LIN {X 0,Y 328.943,Z 502.897,A -85,B 0,C 180,E1 -15636.784,E2 -15636.784} C_VEL
LIN {X 0,Y 327.301,Z 513.257,A -85,B 0,C 180,E1 -15637.783,E2 -15637.783} C_VEL
LIN {X 0,Y 325.235,Z 524.397,A -85,B 0,C 180,E1 -15639.111,E2 -15639.111} C_VEL
LIN {X 0,Y 323.008,Z 534.604,A -85,B 0,C 180,E1 -15640.621,E2 -15640.621} C_VEL
LIN {X 0,Y 320.683,Z 544.507,A -85,B 0,C 180,E1 -15642.462,E2 -15642.462} C_VEL
LIN {X 0,Y 318.696,Z 552.395,A -85,B 0,C 180,E1 -15644.327,E2 -15644.327} C_VEL
LIN {X 0,Y 317.23,Z 557.815,A -85,B 0,C 180,E1 -15645.895,E2 -15645.895} C_VEL
LIN {X 0,Y 315.687,Z 563.068,A -85,B 0,C 180,E1 -15647.79,E2 -15647.79} C_VEL
LIN {X 0,Y 314.434,Z 567.146,A -85,B 0,C 180,E1 -15649.699,E2 -15649.699} C_VEL
LIN {X 0,Y 313.55,Z 569.293,A -85,B 0,C 180,E1 -15650.973,E2 -15650.973} C_VEL
LIN {X 0,Y 313.019,Z 570.939,A -85,B 0,C 180,E1 -15652.258,E2 -15652.258} C_VEL
LIN {X 0,Y 312.547,Z 572.122,A -85,B 0,C 180,E1 -15653.544,E2 -15653.544} C_VEL
LIN {X 0,Y 312.335,Z 572.873,A -85,B 0,C 180,E1 -15654.836,E2 -15654.836} C_VEL
LIN {X 0,Y 312.032,Z 573.237,A -85,B 0,C 180,E1 -15656.125,E2 -15656.125} C_VEL
LIN {X 0,Y 311.617,Z 573.155,A -85,B 0,C 180,E1 -15657.415,E2 -15657.415} C_VEL
LIN {X 0,Y 311.355,Z 572.635,A -85,B 0,C 180,E1 -15658.706,E2 -15658.706} C_VEL
LIN {X 0,Y 311.243,Z 571.699,A -85,B 0,C 180,E1 -15660,E2 -15660} C_VEL
LIN {X 0,Y 311.196,Z 570.316,A -85,B 0,C 180,E1 -15661.294,E2 -15661.294} C_VEL
LIN {X 0,Y 311.223,Z 567.384,A -85,B 0,C 180,E1 -15663.236,E2 -15663.236} C_VEL
LIN {X 0,Y 311.418,Z 563.364,A -85,B 0,C 180,E1 -15665.179,E2 -15665.179} C_VEL
LIN {X 0,Y 311.687,Z 557.186,A -85,B 0,C 180,E1 -15667.436,E2 -15667.436} C_VEL
LIN {X 0,Y 312.083,Z 550.339,A -85,B 0,C 180,E1 -15669.396,E2 -15669.396} C_VEL
LIN {X 0,Y 312.706,Z 541.811,A -85,B 0,C 180,E1 -15671.341,E2 -15671.341} C_VEL
LIN {X 0,Y 313.329,Z 533.139,A -85,B 0,C 180,E1 -15672.962,E2 -15672.962} C_VEL
LIN {X 0,Y 314.181,Z 522.592,A -85,B 0,C 180,E1 -15674.575,E2 -15674.575} C_VEL
LIN {X 0,Y 315.066,Z 510.768,A -85,B 0,C 180,E1 -15676.027,E2 -15676.027} C_VEL
LIN {X 0,Y 315.637,Z 499.309,A -85,B 0,C 180,E1 -15677.159,E2 -15677.159} C_VEL
LIN {X 0,Y 316.398,Z 485.475,A -85,B 0,C 180,E1 -15678.202,E2 -15678.202} C_VEL
LIN {X 0,Y 317.017,Z 472.382,A -85,B 0,C 180,E1 -15678.918,E2 -15678.918} C_VEL
LIN {X 0,Y 317.51,Z 455.689,A -85,B 0,C 180,E1 -15679.517,E2 -15679.517} C_VEL
LIN {X 0,Y 319.541,Z 389.489,A -85,B 0,C 180,E1 -15681.639,E2 -15681.639} C_VEL
LIN {X 0,Y 312.571,Z 367.548,A -85,B 0,C 180,E1 -15682.686,E2 -15682.686} C_VEL
LIN {X 0,Y 312.608,Z 367.544,A -85,B 0,C 180,E1 -15685.935,E2 -15685.935} C_VEL
LIN {X 0,Y 312.55,Z 367.55,A -85,B 0,C 180,E1 -15689.649,E2 -15689.649} C_VEL
LIN {X 0,Y 312.524,Z 367.553,A -85,B 0,C 180,E1 -15693.688,E2 -15693.688} C_VEL
LIN {X 0,Y 312.53,Z 367.552,A -85,B 0,C 180,E1 -15697.384,E2 -15697.384} C_VEL
LIN {X 0,Y 312.494,Z 367.558,A -85,B 0,C 180,E1 -15700.708,E2 -15700.708} C_VEL
LIN {X 0,Y 312.456,Z 367.566,A -85,B 0,C 180,E1 -15704.209,E2 -15704.209} C_VEL
LIN {X 0,Y 312.488,Z 367.56,A -85,B 0,C 180,E1 -15707.918,E2 -15707.918} C_VEL
LIN {X 0,Y 312.539,Z 367.553,A -85,B 0,C 180,E1 -15711.91,E2 -15711.91} C_VEL
LIN {X 0,Y 312.51,Z 367.556,A -85,B 0,C 180,E1 -15715.789,E2 -15715.789} C_VEL
LIN {X 0,Y 312.524,Z 367.553,A -85,B 0,C 180,E1 -15718.853,E2 -15718.853} C_VEL
LIN {X 0,Y 312.574,Z 367.549,A -85,B 0,C 180,E1 -15721.823,E2 -15721.823} C_VEL
LIN {X 0,Y 312.589,Z 367.545,A -85,B 0,C 180,E1 -15724.71,E2 -15724.71} C_VEL
LIN {X 0,Y 312.591,Z 367.545,A -85,B 0,C 180,E1 -15727.528,E2 -15727.528} C_VEL
LIN {X 0,Y 312.642,Z 367.54,A -85,B 0,C 180,E1 -15731.655,E2 -15731.655} C_VEL
LIN {X 0,Y 312.697,Z 367.533,A -85,B 0,C 180,E1 -15735.685,E2 -15735.685} C_VEL
LIN {X 0,Y 312.701,Z 367.532,A -85,B 0,C 180,E1 -15739.64,E2 -15739.64} C_VEL
LIN {X 0,Y 312.855,Z 367.515,A -85,B 0,C 180,E1 -15742.252,E2 -15742.252} C_VEL
LIN {X 0,Y 312.718,Z 367.528,A -85,B 0,C 180,E1 -15744.841,E2 -15744.841} C_VEL
LIN {X 0,Y 312.993,Z 367.495,A -85,B 0,C 180,E1 -15748.712,E2 -15748.712} C_VEL
LIN {X 0,Y 313.122,Z 367.484,A -85,B 0,C 180,E1 -15749.999,E2 -15749.999} C_VEL
LIN {X 0,Y 312.94,Z 367.502,A -85,B 0,C 180,E1 -15752.573,E2 -15752.573} C_VEL
LIN {X 0,Y 312.911,Z 367.506,A -85,B 0,C 180,E1 -15756.446,E2 -15756.446} C_VEL
LIN {X 0,Y 312.787,Z 367.52,A -85,B 0,C 180,E1 -15759.048,E2 -15759.048} C_VEL
LIN {X 0,Y 312.633,Z 367.539,A -85,B 0,C 180,E1 -15762.989,E2 -15762.989} C_VEL
LIN {X 0,Y 312.637,Z 367.541,A -85,B 0,C 180,E1 -15765.648,E2 -15765.648} C_VEL
LIN {X 0,Y 312.629,Z 367.54,A -85,B 0,C 180,E1 -15769.235,E2 -15769.235} C_VEL
LIN {X 0,Y 312.543,Z 367.55,A -85,B 0,C 180,E1 -15772.788,E2 -15772.788} C_VEL
LIN {X 0,Y 312.6,Z 367.548,A -85,B 0,C 180,E1 -15775.934,E2 -15775.934} C_VEL
LIN {X 0,Y 312.542,Z 367.554,A -85,B 0,C 180,E1 -15779.648,E2 -15779.648} C_VEL
LIN {X 0,Y 312.515,Z 367.558,A -85,B 0,C 180,E1 -15783.688,E2 -15783.688} C_VEL
LIN {X 0,Y 312.548,Z 367.551,A -85,B 0,C 180,E1 -15787.38,E2 -15787.38} C_VEL
LIN {X 0,Y 312.529,Z 367.552,A -85,B 0,C 180,E1 -15790.701,E2 -15790.701} C_VEL
LIN {X 0,Y 312.589,Z 367.546,A -85,B 0,C 180,E1 -15794.183,E2 -15794.183} C_VEL
LIN {X 0,Y 312.55,Z 367.553,A -85,B 0,C 180,E1 -15797.903,E2 -15797.903} C_VEL
LIN {X 0,Y 312.55,Z 367.553,A -85,B 0,C 180,E1 -15801.904,E2 -15801.904} C_VEL
LIN {X 0,Y 312.498,Z 367.56,A -85,B 0,C 180,E1 -15805.789,E2 -15805.789} C_VEL
LIN {X 0,Y 312.515,Z 367.554,A -85,B 0,C 180,E1 -15808.853,E2 -15808.853} C_VEL
LIN {X 0,Y 312.576,Z 367.55,A -85,B 0,C 180,E1 -15811.825,E2 -15811.825} C_VEL
LIN {X 0,Y 312.577,Z 367.546,A -85,B 0,C 180,E1 -15814.71,E2 -15814.71} C_VEL
LIN {X 0,Y 312.578,Z 367.55,A -85,B 0,C 180,E1 -15817.528,E2 -15817.528} C_VEL
LIN {X 0,Y 312.616,Z 367.542,A -85,B 0,C 180,E1 -15821.173,E2 -15821.173} C_VEL
LIN {X 0,Y 311.964,Z 367.628,A -85,B 0,C 180,E1 -15822.249,E2 -15822.249} C_VEL
LIN {X 0,Y 309.133,Z 367.983,A -85,B 0,C 180,E1 -15824.002,E2 -15824.002} C_VEL
LIN {X 0,Y 306.716,Z 368.281,A -85,B 0,C 180,E1 -15825.423,E2 -15825.423} C_VEL
LIN {X 0,Y 305.666,Z 368.407,A -85,B 0,C 180,E1 -15826.523,E2 -15826.523} C_VEL
LIN {X 0,Y 305.573,Z 368.417,A -85,B 0,C 180,E1 -15826.895,E2 -15826.895} C_VEL
LIN {X 0,Y 305.787,Z 368.394,A -85,B 0,C 180,E1 -15831.208,E2 -15831.208} C_VEL
LIN {X 0,Y 305.843,Z 368.389,A -85,B 0,C 180,E1 -15833.403,E2 -15833.403} C_VEL
LIN {X 0,Y 305.89,Z 368.383,A -85,B 0,C 180,E1 -15837.366,E2 -15837.366} C_VEL
LIN {X 0,Y 306.064,Z 368.358,A -85,B 0,C 180,E1 -15840,E2 -15840} C_VEL
LIN {X 0,Y 305.879,Z 368.38,A -85,B 0,C 180,E1 -15842.634,E2 -15842.634} C_VEL
LIN {X 0,Y 305.846,Z 368.385,A -85,B 0,C 180,E1 -15846.598,E2 -15846.598} C_VEL
LIN {X 0,Y 305.727,Z 368.403,A -85,B 0,C 180,E1 -15849.26,E2 -15849.26} C_VEL
LIN {X 0,Y 305.582,Z 368.421,A -85,B 0,C 180,E1 -15853.296,E2 -15853.296} C_VEL
LIN {X 0,Y 305.585,Z 368.418,A -85,B 0,C 180,E1 -15856.021,E2 -15856.021} C_VEL
LIN {X 0,Y 305.568,Z 368.424,A -85,B 0,C 180,E1 -15859.446,E2 -15859.446} C_VEL
LIN {X 0,Y 305.482,Z 368.432,A -85,B 0,C 180,E1 -15863.042,E2 -15863.042} C_VEL
LIN {X 0,Y 305.517,Z 368.425,A -85,B 0,C 180,E1 -15866.22,E2 -15866.22} C_VEL
LIN {X 0,Y 305.48,Z 368.432,A -85,B 0,C 180,E1 -15869.048,E2 -15869.048} C_VEL
LIN {X 0,Y 305.434,Z 368.437,A -85,B 0,C 180,E1 -15871.954,E2 -15871.954} C_VEL
LIN {X 0,Y 305.456,Z 368.437,A -85,B 0,C 180,E1 -15875.114,E2 -15875.114} C_VEL
LIN {X 0,Y 305.489,Z 368.429,A -85,B 0,C 180,E1 -15878.541,E2 -15878.541} C_VEL
LIN {X 0,Y 305.516,Z 368.426,A -85,B 0,C 180,E1 -15882.601,E2 -15882.601} C_VEL
LIN {X 0,Y 305.529,Z 368.423,A -85,B 0,C 180,E1 -15886.366,E2 -15886.366} C_VEL
LIN {X 0,Y 305.495,Z 368.429,A -85,B 0,C 180,E1 -15889.901,E2 -15889.901} C_VEL
LIN {X 0,Y 305.498,Z 368.429,A -85,B 0,C 180,E1 -15893.628,E2 -15893.628} C_VEL
LIN {X 0,Y 305.54,Z 368.505,A -85,B 0,C 180,E1 -15896.939,E2 -15896.939} C_VEL
LIN {X 0,Y 308.728,Z 384.104,A -85,B 0,C 180,E1 -15901.072,E2 -15901.072} C_VEL
LIN {X 0,Y 309.707,Z 390.276,A -85,B 0,C 180,E1 -15902.649,E2 -15902.649} C_VEL
LIN {X 0,Y 308.052,Z 404.751,A -85,B 0,C 180,E1 -15906.14,E2 -15906.14} C_VEL
LIN {X 0,Y 307.818,Z 407.252,A -85,B 0,C 180,E1 -15906.719,E2 -15906.719} C_VEL
LIN {X 0,Y 309.835,Z 432.681,A -85,B 0,C 180,E1 -15907.693,E2 -15907.693} C_VEL
LIN {X 0,Y 311.778,Z 451.87,A -85,B 0,C 180,E1 -15908.433,E2 -15908.433} C_VEL
LIN {X 0,Y 309.786,Z 517.337,A -85,B 0,C 180,E1 -15910.667,E2 -15910.667} C_VEL
LIN {X 0,Y 309.008,Z 530.335,A -85,B 0,C 180,E1 -15911.349,E2 -15911.349} C_VEL
LIN {X 0,Y 308.149,Z 542.629,A -85,B 0,C 180,E1 -15912.241,E2 -15912.241} C_VEL
LIN {X 0,Y 307.335,Z 554.72,A -85,B 0,C 180,E1 -15913.392,E2 -15913.392} C_VEL
LIN {X 0,Y 306.479,Z 565.586,A -85,B 0,C 180,E1 -15914.687,E2 -15914.687} C_VEL
LIN {X 0,Y 305.7,Z 575.858,A -85,B 0,C 180,E1 -15916.202,E2 -15916.202} C_VEL
LIN {X 0,Y 304.994,Z 585.89,A -85,B 0,C 180,E1 -15918.032,E2 -15918.032} C_VEL
LIN {X 0,Y 304.522,Z 593.338,A -85,B 0,C 180,E1 -15919.698,E2 -15919.698} C_VEL
LIN {X 0,Y 304.314,Z 600.602,A -85,B 0,C 180,E1 -15921.702,E2 -15921.702} C_VEL
LIN {X 0,Y 304.237,Z 606.711,A -85,B 0,C 180,E1 -15923.857,E2 -15923.857} C_VEL
LIN {X 0,Y 304.227,Z 611.32,A -85,B 0,C 180,E1 -15926.028,E2 -15926.028} C_VEL
LIN {X 0,Y 304.239,Z 613.406,A -85,B 0,C 180,E1 -15927.354,E2 -15927.354} C_VEL
LIN {X 0,Y 304.424,Z 615.02,A -85,B 0,C 180,E1 -15928.679,E2 -15928.679} C_VEL
LIN {X 0,Y 304.4,Z 616.15,A -85,B 0,C 180,E1 -15930.002,E2 -15930.002} C_VEL
LIN {X 0,Y 304.147,Z 616.77,A -85,B 0,C 180,E1 -15931.326,E2 -15931.326} C_VEL
LIN {X 0,Y 304.008,Z 616.934,A -85,B 0,C 180,E1 -15932.652,E2 -15932.652} C_VEL
LIN {X 0,Y 303.856,Z 616.667,A -85,B 0,C 180,E1 -15933.98,E2 -15933.98} C_VEL
LIN {X 0,Y 303.815,Z 615.504,A -85,B 0,C 180,E1 -15935.901,E2 -15935.901} C_VEL
LIN {X 0,Y 304.016,Z 612.303,A -85,B 0,C 180,E1 -15938.644,E2 -15938.644} C_VEL
LIN {X 0,Y 304.52,Z 608.766,A -85,B 0,C 180,E1 -15940.641,E2 -15940.641} C_VEL
LIN {X 0,Y 305.392,Z 604.144,A -85,B 0,C 180,E1 -15942.63,E2 -15942.63} C_VEL
LIN {X 0,Y 306.856,Z 597.249,A -85,B 0,C 180,E1 -15944.933,E2 -15944.933} C_VEL
LIN {X 0,Y 308.362,Z 590.584,A -85,B 0,C 180,E1 -15946.723,E2 -15946.723} C_VEL
LIN {X 0,Y 310.363,Z 582.557,A -85,B 0,C 180,E1 -15948.484,E2 -15948.484} C_VEL
LIN {X 0,Y 312.535,Z 573.888,A -85,B 0,C 180,E1 -15950.057,E2 -15950.057} C_VEL
LIN {X 0,Y 314.949,Z 563.526,A -85,B 0,C 180,E1 -15951.606,E2 -15951.606} C_VEL
LIN {X 0,Y 317.789,Z 550.815,A -85,B 0,C 180,E1 -15953.114,E2 -15953.114} C_VEL
LIN {X 0,Y 320.028,Z 539.948,A -85,B 0,C 180,E1 -15954.144,E2 -15954.144} C_VEL
LIN {X 0,Y 322.595,Z 526.17,A -85,B 0,C 180,E1 -15955.141,E2 -15955.141} C_VEL
LIN {X 0,Y 324.642,Z 512.058,A -85,B 0,C 180,E1 -15955.916,E2 -15955.916} C_VEL
LIN {X 0,Y 328.062,Z 476.175,A -85,B 0,C 180,E1 -15957.317,E2 -15957.317} C_VEL
LIN {X 0,Y 329.941,Z 456.205,A -85,B 0,C 180,E1 -15958.101,E2 -15958.101} C_VEL
LIN {X 0,Y 329.581,Z 444.672,A -85,B 0,C 180,E1 -15958.851,E2 -15958.851} C_VEL
LIN {X 0,Y 328.161,Z 430.684,A -85,B 0,C 180,E1 -15960.026,E2 -15960.026} C_VEL
LIN {X 0,Y 326.387,Z 418.697,A -85,B 0,C 180,E1 -15961.253,E2 -15961.253} C_VEL
LIN {X 0,Y 325.891,Z 416.427,A -85,B 0,C 180,E1 -15961.54,E2 -15961.54} C_VEL
LIN {X 0,Y 323.766,Z 411.453,A -85,B 0,C 180,E1 -15962.48,E2 -15962.48} C_VEL
LIN {X 0,Y 320.896,Z 405.401,A -85,B 0,C 180,E1 -15963.838,E2 -15963.838} C_VEL
LIN {X 0,Y 317.423,Z 398.46,A -85,B 0,C 180,E1 -15965.73,E2 -15965.73} C_VEL
LIN {X 0,Y 312.795,Z 390.131,A -85,B 0,C 180,E1 -15969.007,E2 -15969.007} C_VEL
LIN {X 0,Y 311.626,Z 386.594,A -85,B 0,C 180,E1 -15971.906,E2 -15971.906} C_VEL
LIN {X 0,Y 310.903,Z 384.372,A -85,B 0,C 180,E1 -15974.489,E2 -15974.489} C_VEL
LIN {X 0,Y 310.476,Z 382.906,A -85,B 0,C 180,E1 -15977.227,E2 -15977.227} C_VEL
LIN {X 0,Y 310.416,Z 382.585,A -85,B 0,C 180,E1 -15979.115,E2 -15979.115} C_VEL
LIN {X 0,Y 313.495,Z 385.341,A -85,B 0,C 180,E1 -15982.4,E2 -15982.4} C_VEL
LIN {X 0,Y 314.523,Z 386.096,A -85,B 0,C 180,E1 -15983.135,E2 -15983.135} C_VEL
LIN {X 0,Y 317.228,Z 389.292,A -85,B 0,C 180,E1 -15984.908,E2 -15984.908} C_VEL
LIN {X 0,Y 318.425,Z 390.623,A -85,B 0,C 180,E1 -15985.572,E2 -15985.572} C_VEL
LIN {X 0,Y 321.705,Z 394.693,A -85,B 0,C 180,E1 -15987.201,E2 -15987.201} C_VEL
LIN {X 0,Y 324.633,Z 398.637,A -85,B 0,C 180,E1 -15988.465,E2 -15988.465} C_VEL
LIN {X 0,Y 327.692,Z 403.121,A -85,B 0,C 180,E1 -15989.668,E2 -15989.668} C_VEL
LIN {X 0,Y 331.656,Z 409.714,A -85,B 0,C 180,E1 -15991.09,E2 -15991.09} C_VEL
LIN {X 0,Y 333.388,Z 413.263,A -85,B 0,C 180,E1 -15991.699,E2 -15991.699} C_VEL
LIN {X 0,Y 326.897,Z 475.924,A -85,B 0,C 180,E1 -15994.149,E2 -15994.149} C_VEL
LIN {X 0,Y 325.559,Z 488.663,A -85,B 0,C 180,E1 -15994.849,E2 -15994.849} C_VEL
LIN {X 0,Y 323.853,Z 501.404,A -85,B 0,C 180,E1 -15995.794,E2 -15995.794} C_VEL
LIN {X 0,Y 321.752,Z 513.792,A -85,B 0,C 180,E1 -15996.981,E2 -15996.981} C_VEL
LIN {X 0,Y 319.479,Z 525.285,A -85,B 0,C 180,E1 -15998.378,E2 -15998.378} C_VEL
LIN {X 0,Y 317.114,Z 535.398,A -85,B 0,C 180,E1 -15999.909,E2 -15999.909} C_VEL
LIN {X 0,Y 314.612,Z 545.241,A -85,B 0,C 180,E1 -16001.775,E2 -16001.775} C_VEL
LIN {X 0,Y 312.434,Z 553.103,A -85,B 0,C 180,E1 -16003.669,E2 -16003.669} C_VEL
LIN {X 0,Y 310.538,Z 559.458,A -85,B 0,C 180,E1 -16005.585,E2 -16005.585} C_VEL
LIN {X 0,Y 308.907,Z 564.501,A -85,B 0,C 180,E1 -16007.518,E2 -16007.518} C_VEL
LIN {X 0,Y 307.57,Z 568.385,A -85,B 0,C 180,E1 -16009.467,E2 -16009.467} C_VEL
LIN {X 0,Y 306.649,Z 570.41,A -85,B 0,C 180,E1 -16010.768,E2 -16010.768} C_VEL
LIN {X 0,Y 306.06,Z 571.917,A -85,B 0,C 180,E1 -16012.081,E2 -16012.081} C_VEL
LIN {X 0,Y 305.554,Z 573.011,A -85,B 0,C 180,E1 -16013.396,E2 -16013.396} C_VEL
LIN {X 0,Y 305.31,Z 573.673,A -85,B 0,C 180,E1 -16014.717,E2 -16014.717} C_VEL
LIN {X 0,Y 304.98,Z 573.9,A -85,B 0,C 180,E1 -16016.036,E2 -16016.036} C_VEL
LIN {X 0,Y 304.562,Z 573.716,A -85,B 0,C 180,E1 -16017.355,E2 -16017.355} C_VEL
LIN {X 0,Y 304.294,Z 573.113,A -85,B 0,C 180,E1 -16018.676,E2 -16018.676} C_VEL
LIN {X 0,Y 304.182,Z 572.069,A -85,B 0,C 180,E1 -16020,E2 -16020} C_VEL
LIN {X 0,Y 304.101,Z 570.559,A -85,B 0,C 180,E1 -16021.324,E2 -16021.324} C_VEL
LIN {X 0,Y 304.139,Z 567.466,A -85,B 0,C 180,E1 -16023.312,E2 -16023.312} C_VEL
LIN {X 0,Y 304.338,Z 563.277,A -85,B 0,C 180,E1 -16025.3,E2 -16025.3} C_VEL
LIN {X 0,Y 304.614,Z 557.169,A -85,B 0,C 180,E1 -16027.521,E2 -16027.521} C_VEL
LIN {X 0,Y 305.049,Z 549.774,A -85,B 0,C 180,E1 -16029.615,E2 -16029.615} C_VEL
LIN {X 0,Y 305.698,Z 541.01,A -85,B 0,C 180,E1 -16031.605,E2 -16031.605} C_VEL
LIN {X 0,Y 306.458,Z 531.045,A -85,B 0,C 180,E1 -16033.426,E2 -16033.426} C_VEL
LIN {X 0,Y 307.306,Z 519.872,A -85,B 0,C 180,E1 -16035.078,E2 -16035.078} C_VEL
LIN {X 0,Y 308.09,Z 509.65,A -85,B 0,C 180,E1 -16036.303,E2 -16036.303} C_VEL
LIN {X 0,Y 308.792,Z 496.587,A -85,B 0,C 180,E1 -16037.552,E2 -16037.552} C_VEL
LIN {X 0,Y 309.467,Z 484.356,A -85,B 0,C 180,E1 -16038.453,E2 -16038.453} C_VEL
LIN {X 0,Y 310.003,Z 470.437,A -85,B 0,C 180,E1 -16039.191,E2 -16039.191} C_VEL
LIN {X 0,Y 312.585,Z 390.891,A -85,B 0,C 180,E1 -16041.869,E2 -16041.869} C_VEL
LIN {X 0,Y 305.523,Z 368.424,A -85,B 0,C 180,E1 -16042.982,E2 -16042.982} C_VEL
LIN {X 0,Y 305.553,Z 368.425,A -85,B 0,C 180,E1 -16046.226,E2 -16046.226} C_VEL
LIN {X 0,Y 305.501,Z 368.428,A -85,B 0,C 180,E1 -16049.049,E2 -16049.049} C_VEL
LIN {X 0,Y 305.449,Z 368.436,A -85,B 0,C 180,E1 -16051.951,E2 -16051.951} C_VEL
LIN {X 0,Y 305.467,Z 368.432,A -85,B 0,C 180,E1 -16055.112,E2 -16055.112} C_VEL
LIN {X 0,Y 305.472,Z 368.434,A -85,B 0,C 180,E1 -16058.532,E2 -16058.532} C_VEL
LIN {X 0,Y 305.46,Z 368.435,A -85,B 0,C 180,E1 -16062.585,E2 -16062.585} C_VEL
LIN {X 0,Y 305.43,Z 368.441,A -85,B 0,C 180,E1 -16066.344,E2 -16066.344} C_VEL
LIN {X 0,Y 305.462,Z 368.434,A -85,B 0,C 180,E1 -16069.891,E2 -16069.891} C_VEL
LIN {X 0,Y 305.488,Z 368.43,A -85,B 0,C 180,E1 -16073.63,E2 -16073.63} C_VEL
LIN {X 0,Y 305.469,Z 368.434,A -85,B 0,C 180,E1 -16076.482,E2 -16076.482} C_VEL
LIN {X 0,Y 305.462,Z 368.433,A -85,B 0,C 180,E1 -16079.589,E2 -16079.589} C_VEL
LIN {X 0,Y 305.522,Z 368.426,A -85,B 0,C 180,E1 -16082.607,E2 -16082.607} C_VEL
LIN {X 0,Y 305.512,Z 368.427,A -85,B 0,C 180,E1 -16085.538,E2 -16085.538} C_VEL
LIN {X 0,Y 305.523,Z 368.427,A -85,B 0,C 180,E1 -16089.814,E2 -16089.814} C_VEL
LIN {X 0,Y 305.578,Z 368.419,A -85,B 0,C 180,E1 -16092.602,E2 -16092.602} C_VEL
LIN {X 0,Y 305.652,Z 368.409,A -85,B 0,C 180,E1 -16095.348,E2 -16095.348} C_VEL
LIN {X 0,Y 305.638,Z 368.411,A -85,B 0,C 180,E1 -16099.398,E2 -16099.398} C_VEL
LIN {X 0,Y 305.799,Z 368.396,A -85,B 0,C 180,E1 -16102.073,E2 -16102.073} C_VEL
LIN {X 0,Y 305.689,Z 368.404,A -85,B 0,C 180,E1 -16104.722,E2 -16104.722} C_VEL
LIN {X 0,Y 305.959,Z 368.371,A -85,B 0,C 180,E1 -16108.682,E2 -16108.682} C_VEL
LIN {X 0,Y 305.959,Z 368.371,A -85,B 0,C 180,E1 -16111.315,E2 -16111.315} C_VEL
LIN {X 0,Y 305.853,Z 368.384,A -85,B 0,C 180,E1 -16116.596,E2 -16116.596} C_VEL
LIN {X 0,Y 305.735,Z 368.399,A -85,B 0,C 180,E1 -16119.258,E2 -16119.258} C_VEL
LIN {X 0,Y 305.588,Z 368.417,A -85,B 0,C 180,E1 -16123.294,E2 -16123.294} C_VEL
LIN {X 0,Y 305.593,Z 368.421,A -85,B 0,C 180,E1 -16126.018,E2 -16126.018} C_VEL
LIN {X 0,Y 305.575,Z 368.42,A -85,B 0,C 180,E1 -16129.444,E2 -16129.444} C_VEL
LIN {X 0,Y 305.488,Z 368.429,A -85,B 0,C 180,E1 -16133.04,E2 -16133.04} C_VEL
LIN {X 0,Y 305.544,Z 368.424,A -85,B 0,C 180,E1 -16136.226,E2 -16136.226} C_VEL
LIN {X 0,Y 305.492,Z 368.428,A -85,B 0,C 180,E1 -16139.049,E2 -16139.049} C_VEL
LIN {X 0,Y 305.444,Z 368.439,A -85,B 0,C 180,E1 -16141.95,E2 -16141.95} C_VEL
LIN {X 0,Y 305.458,Z 368.433,A -85,B 0,C 180,E1 -16145.112,E2 -16145.112} C_VEL
LIN {X 0,Y 305.489,Z 368.429,A -85,B 0,C 180,E1 -16148.538,E2 -16148.538} C_VEL
LIN {X 0,Y 305.516,Z 368.426,A -85,B 0,C 180,E1 -16152.598,E2 -16152.598} C_VEL
LIN {X 0,Y 305.528,Z 368.425,A -85,B 0,C 180,E1 -16156.363,E2 -16156.363} C_VEL
LIN {X 0,Y 305.493,Z 368.432,A -85,B 0,C 180,E1 -16159.898,E2 -16159.898} C_VEL
LIN {X 0,Y 305.494,Z 368.433,A -85,B 0,C 180,E1 -16163.625,E2 -16163.625} C_VEL
LIN {X 0,Y 305.457,Z 368.433,A -85,B 0,C 180,E1 -16166.482,E2 -16166.482} C_VEL
LIN {X 0,Y 305.494,Z 368.429,A -85,B 0,C 180,E1 -16170.947,E2 -16170.947} C_VEL
LIN {X 0,Y 305.563,Z 368.421,A -85,B 0,C 180,E1 -16174.087,E2 -16174.087} C_VEL
LIN {X 0,Y 305.492,Z 368.429,A -85,B 0,C 180,E1 -16178.402,E2 -16178.402} C_VEL
LIN {X 0,Y 305.581,Z 368.42,A -85,B 0,C 180,E1 -16181.217,E2 -16181.217} C_VEL
LIN {X 0,Y 305.64,Z 368.413,A -85,B 0,C 180,E1 -16185.349,E2 -16185.349} C_VEL
LIN {X 0,Y 305.573,Z 368.417,A -85,B 0,C 180,E1 -16186.895,E2 -16186.895} C_VEL
LIN {X 0,Y 304.902,Z 368.505,A -85,B 0,C 180,E1 -16187.997,E2 -16187.997} C_VEL
LIN {X 0,Y 302.114,Z 368.853,A -85,B 0,C 180,E1 -16189.793,E2 -16189.793} C_VEL
LIN {X 0,Y 299.784,Z 369.142,A -85,B 0,C 180,E1 -16191.25,E2 -16191.25} C_VEL
LIN {X 0,Y 298.817,Z 369.26,A -85,B 0,C 180,E1 -16192.376,E2 -16192.376} C_VEL
LIN {X 0,Y 298.755,Z 369.267,A -85,B 0,C 180,E1 -16192.757,E2 -16192.757} C_VEL
LIN {X 0,Y 298.839,Z 369.261,A -85,B 0,C 180,E1 -16197.304,E2 -16197.304} C_VEL
LIN {X 0,Y 299.017,Z 369.236,A -85,B 0,C 180,E1 -16200,E2 -16200} C_VEL
LIN {X 0,Y 298.83,Z 369.258,A -85,B 0,C 180,E1 -16202.696,E2 -16202.696} C_VEL
LIN {X 0,Y 298.791,Z 369.264,A -85,B 0,C 180,E1 -16206.754,E2 -16206.754} C_VEL
LIN {X 0,Y 298.672,Z 369.283,A -85,B 0,C 180,E1 -16209.481,E2 -16209.481} C_VEL
LIN {X 0,Y 298.545,Z 369.298,A -85,B 0,C 180,E1 -16213.616,E2 -16213.616} C_VEL
LIN {X 0,Y 298.54,Z 369.295,A -85,B 0,C 180,E1 -16216.409,E2 -16216.409} C_VEL
LIN {X 0,Y 298.503,Z 369.302,A -85,B 0,C 180,E1 -16219.656,E2 -16219.656} C_VEL
LIN {X 0,Y 298.449,Z 369.309,A -85,B 0,C 180,E1 -16223.599,E2 -16223.599} C_VEL
LIN {X 0,Y 298.477,Z 369.302,A -85,B 0,C 180,E1 -16226.576,E2 -16226.576} C_VEL
LIN {X 0,Y 298.408,Z 369.313,A -85,B 0,C 180,E1 -16229.643,E2 -16229.643} C_VEL
LIN {X 0,Y 298.387,Z 369.315,A -85,B 0,C 180,E1 -16232.801,E2 -16232.801} C_VEL
LIN {X 0,Y 298.465,Z 369.305,A -85,B 0,C 180,E1 -16236.815,E2 -16236.815} C_VEL
LIN {X 0,Y 298.451,Z 369.31,A -85,B 0,C 180,E1 -16241.105,E2 -16241.105} C_VEL
LIN {X 0,Y 298.484,Z 369.305,A -85,B 0,C 180,E1 -16245.062,E2 -16245.062} C_VEL
LIN {X 0,Y 298.452,Z 369.308,A -85,B 0,C 180,E1 -16248.899,E2 -16248.899} C_VEL
LIN {X 0,Y 298.466,Z 369.309,A -85,B 0,C 180,E1 -16253.188,E2 -16253.188} C_VEL
LIN {X 0,Y 298.496,Z 369.486,A -85,B 0,C 180,E1 -16256.762,E2 -16256.762} C_VEL
LIN {X 0,Y 301.742,Z 385.347,A -85,B 0,C 180,E1 -16261.064,E2 -16261.064} C_VEL
LIN {X 0,Y 302.621,Z 390.142,A -85,B 0,C 180,E1 -16262.326,E2 -16262.326} C_VEL
LIN {X 0,Y 301.575,Z 400.254,A -85,B 0,C 180,E1 -16264.832,E2 -16264.832} C_VEL
LIN {X 0,Y 300.829,Z 406.644,A -85,B 0,C 180,E1 -16266.405,E2 -16266.405} C_VEL
LIN {X 0,Y 302.792,Z 432.618,A -85,B 0,C 180,E1 -16267.435,E2 -16267.435} C_VEL
LIN {X 0,Y 304.777,Z 452.461,A -85,B 0,C 180,E1 -16268.22,E2 -16268.22} C_VEL
LIN {X 0,Y 302.754,Z 517.001,A -85,B 0,C 180,E1 -16270.509,E2 -16270.509} C_VEL
LIN {X 0,Y 301.945,Z 530.531,A -85,B 0,C 180,E1 -16271.248,E2 -16271.248} C_VEL
LIN {X 0,Y 301.08,Z 542.588,A -85,B 0,C 180,E1 -16272.161,E2 -16272.161} C_VEL
LIN {X 0,Y 300.244,Z 554.573,A -85,B 0,C 180,E1 -16273.339,E2 -16273.339} C_VEL
LIN {X 0,Y 299.437,Z 564.734,A -85,B 0,C 180,E1 -16274.58,E2 -16274.58} C_VEL
LIN {X 0,Y 298.636,Z 574.547,A -85,B 0,C 180,E1 -16276.043,E2 -16276.043} C_VEL
LIN {X 0,Y 297.995,Z 583.857,A -85,B 0,C 180,E1 -16277.747,E2 -16277.747} C_VEL
LIN {X 0,Y 297.458,Z 592.944,A -85,B 0,C 180,E1 -16279.795,E2 -16279.795} C_VEL
LIN {X 0,Y 297.27,Z 600.157,A -85,B 0,C 180,E1 -16281.847,E2 -16281.847} C_VEL
LIN {X 0,Y 297.191,Z 605.653,A -85,B 0,C 180,E1 -16283.818,E2 -16283.818} C_VEL
LIN {X 0,Y 297.192,Z 610.177,A -85,B 0,C 180,E1 -16285.933,E2 -16285.933} C_VEL
LIN {X 0,Y 297.189,Z 612.402,A -85,B 0,C 180,E1 -16287.291,E2 -16287.291} C_VEL
LIN {X 0,Y 297.379,Z 614.101,A -85,B 0,C 180,E1 -16288.647,E2 -16288.647} C_VEL
LIN {X 0,Y 297.355,Z 615.3,A -85,B 0,C 180,E1 -16290.002,E2 -16290.002} C_VEL
LIN {X 0,Y 297.085,Z 616.027,A -85,B 0,C 180,E1 -16291.357,E2 -16291.357} C_VEL
LIN {X 0,Y 296.921,Z 616.297,A -85,B 0,C 180,E1 -16292.715,E2 -16292.715} C_VEL
LIN {X 0,Y 296.781,Z 616.102,A -85,B 0,C 180,E1 -16294.075,E2 -16294.075} C_VEL
LIN {X 0,Y 296.739,Z 615.217,A -85,B 0,C 180,E1 -16295.881,E2 -16295.881} C_VEL
LIN {X 0,Y 296.866,Z 612.977,A -85,B 0,C 180,E1 -16298.168,E2 -16298.168} C_VEL
LIN {X 0,Y 297.293,Z 609.944,A -85,B 0,C 180,E1 -16300.214,E2 -16300.214} C_VEL
LIN {X 0,Y 298.038,Z 605.879,A -85,B 0,C 180,E1 -16302.254,E2 -16302.254} C_VEL
LIN {X 0,Y 299.539,Z 599.701,A -85,B 0,C 180,E1 -16304.611,E2 -16304.611} C_VEL
LIN {X 0,Y 301.199,Z 592.635,A -85,B 0,C 180,E1 -16306.74,E2 -16306.74} C_VEL
LIN {X 0,Y 303.266,Z 585.021,A -85,B 0,C 180,E1 -16308.583,E2 -16308.583} C_VEL
LIN {X 0,Y 305.964,Z 575.175,A -85,B 0,C 180,E1 -16310.507,E2 -16310.507} C_VEL
LIN {X 0,Y 308.774,Z 564.192,A -85,B 0,C 180,E1 -16312.236,E2 -16312.236} C_VEL
LIN {X 0,Y 311.44,Z 553.264,A -85,B 0,C 180,E1 -16313.614,E2 -16313.614} C_VEL
LIN {X 0,Y 313.724,Z 543.116,A -85,B 0,C 180,E1 -16314.662,E2 -16314.662} C_VEL
LIN {X 0,Y 316.579,Z 529.601,A -85,B 0,C 180,E1 -16315.741,E2 -16315.741} C_VEL
LIN {X 0,Y 318.93,Z 515.652,A -85,B 0,C 180,E1 -16316.592,E2 -16316.592} C_VEL
LIN {X 0,Y 320.792,Z 499.774,A -85,B 0,C 180,E1 -16317.305,E2 -16317.305} C_VEL
LIN {X 0,Y 325.081,Z 457.947,A -85,B 0,C 180,E1 -16318.951,E2 -16318.951} C_VEL
LIN {X 0,Y 324.898,Z 447.162,A -85,B 0,C 180,E1 -16319.673,E2 -16319.673} C_VEL
LIN {X 0,Y 323.722,Z 433.569,A -85,B 0,C 180,E1 -16320.858,E2 -16320.858} C_VEL
LIN {X 0,Y 322.171,Z 421.452,A -85,B 0,C 180,E1 -16322.144,E2 -16322.144} C_VEL
LIN {X 0,Y 320.238,Z 416.65,A -85,B 0,C 180,E1 -16323.079,E2 -16323.079} C_VEL
LIN {X 0,Y 317.717,Z 411.031,A -85,B 0,C 180,E1 -16324.381,E2 -16324.381} C_VEL
LIN {X 0,Y 314.611,Z 404.445,A -85,B 0,C 180,E1 -16326.23,E2 -16326.23} C_VEL
LIN {X 0,Y 310.384,Z 396.211,A -85,B 0,C 180,E1 -16329.558,E2 -16329.558} C_VEL
LIN {X 0,Y 308.158,Z 392.537,A -85,B 0,C 180,E1 -16332.309,E2 -16332.309} C_VEL
LIN {X 0,Y 307.36,Z 390.366,A -85,B 0,C 180,E1 -16334.859,E2 -16334.859} C_VEL
LIN {X 0,Y 307.599,Z 389.504,A -85,B 0,C 180,E1 -16336.983,E2 -16336.983} C_VEL
LIN {X 0,Y 308.68,Z 389.511,A -85,B 0,C 180,E1 -16339.149,E2 -16339.149} C_VEL
LIN {X 0,Y 311.883,Z 392.311,A -85,B 0,C 180,E1 -16342.524,E2 -16342.524} C_VEL
LIN {X 0,Y 312.998,Z 393.775,A -85,B 0,C 180,E1 -16343.408,E2 -16343.408} C_VEL
LIN {X 0,Y 315.842,Z 396.909,A -85,B 0,C 180,E1 -16345.191,E2 -16345.191} C_VEL
LIN {X 0,Y 319.066,Z 401.077,A -85,B 0,C 180,E1 -16346.887,E2 -16346.887} C_VEL
LIN {X 0,Y 322.29,Z 405.609,A -85,B 0,C 180,E1 -16348.347,E2 -16348.347} C_VEL
LIN {X 0,Y 325.833,Z 411.201,A -85,B 0,C 180,E1 -16349.786,E2 -16349.786} C_VEL
LIN {X 0,Y 328.573,Z 416.308,A -85,B 0,C 180,E1 -16350.823,E2 -16350.823} C_VEL
LIN {X 0,Y 321.728,Z 478.504,A -85,B 0,C 180,E1 -16353.353,E2 -16353.353} C_VEL
LIN {X 0,Y 320.004,Z 492.71,A -85,B 0,C 180,E1 -16354.206,E2 -16354.206} C_VEL
LIN {X 0,Y 318.154,Z 504.831,A -85,B 0,C 180,E1 -16355.184,E2 -16355.184} C_VEL
LIN {X 0,Y 315.926,Z 516.661,A -85,B 0,C 180,E1 -16356.395,E2 -16356.395} C_VEL
LIN {X 0,Y 313.559,Z 527.416,A -85,B 0,C 180,E1 -16357.776,E2 -16357.776} C_VEL
LIN {X 0,Y 310.829,Z 538.129,A -85,B 0,C 180,E1 -16359.484,E2 -16359.484} C_VEL
LIN {X 0,Y 308.167,Z 547.496,A -85,B 0,C 180,E1 -16361.38,E2 -16361.38} C_VEL
LIN {X 0,Y 305.88,Z 555.053,A -85,B 0,C 180,E1 -16363.309,E2 -16363.309} C_VEL
LIN {X 0,Y 303.874,Z 561.157,A -85,B 0,C 180,E1 -16365.261,E2 -16365.261} C_VEL
LIN {X 0,Y 302.133,Z 565.966,A -85,B 0,C 180,E1 -16367.233,E2 -16367.233} C_VEL
LIN {X 0,Y 300.702,Z 569.639,A -85,B 0,C 180,E1 -16369.223,E2 -16369.223} C_VEL
LIN {X 0,Y 299.749,Z 571.503,A -85,B 0,C 180,E1 -16370.553,E2 -16370.553} C_VEL
LIN {X 0,Y 299.106,Z 572.916,A -85,B 0,C 180,E1 -16371.895,E2 -16371.895} C_VEL
LIN {X 0,Y 298.566,Z 573.91,A -85,B 0,C 180,E1 -16373.241,E2 -16373.241} C_VEL
LIN {X 0,Y 298.274,Z 574.427,A -85,B 0,C 180,E1 -16374.592,E2 -16374.592} C_VEL
LIN {X 0,Y 297.931,Z 574.548,A -85,B 0,C 180,E1 -16375.942,E2 -16375.942} C_VEL
LIN {X 0,Y 297.508,Z 574.274,A -85,B 0,C 180,E1 -16377.292,E2 -16377.292} C_VEL
LIN {X 0,Y 297.236,Z 573.559,A -85,B 0,C 180,E1 -16378.645,E2 -16378.645} C_VEL
LIN {X 0,Y 297.102,Z 572.379,A -85,B 0,C 180,E1 -16380,E2 -16380} C_VEL
LIN {X 0,Y 296.995,Z 569.809,A -85,B 0,C 180,E1 -16382.034,E2 -16382.034} C_VEL
LIN {X 0,Y 297.137,Z 566.188,A -85,B 0,C 180,E1 -16384.069,E2 -16384.069} C_VEL
LIN {X 0,Y 297.285,Z 561.408,A -85,B 0,C 180,E1 -16386.107,E2 -16386.107} C_VEL
LIN {X 0,Y 297.647,Z 555.347,A -85,B 0,C 180,E1 -16388.144,E2 -16388.144} C_VEL
LIN {X 0,Y 298.133,Z 547.794,A -85,B 0,C 180,E1 -16390.183,E2 -16390.183} C_VEL
LIN {X 0,Y 298.83,Z 538.367,A -85,B 0,C 180,E1 -16392.22,E2 -16392.22} C_VEL
LIN {X 0,Y 299.636,Z 528.751,A -85,B 0,C 180,E1 -16393.911,E2 -16393.911} C_VEL
LIN {X 0,Y 300.51,Z 516.785,A -85,B 0,C 180,E1 -16395.602,E2 -16395.602} C_VEL
LIN {X 0,Y 301.281,Z 505.252,A -85,B 0,C 180,E1 -16396.911,E2 -16396.911} C_VEL
LIN {X 0,Y 302.017,Z 492.481,A -85,B 0,C 180,E1 -16398.046,E2 -16398.046} C_VEL
LIN {X 0,Y 302.651,Z 480.181,A -85,B 0,C 180,E1 -16398.884,E2 -16398.884} C_VEL
LIN {X 0,Y 303.115,Z 466.092,A -85,B 0,C 180,E1 -16399.557,E2 -16399.557} C_VEL
LIN {X 0,Y 305.51,Z 391.939,A -85,B 0,C 180,E1 -16402.108,E2 -16402.108} C_VEL
LIN {X 0,Y 298.472,Z 369.301,A -85,B 0,C 180,E1 -16403.252,E2 -16403.252} C_VEL
LIN {X 0,Y 298.495,Z 369.304,A -85,B 0,C 180,E1 -16406.574,E2 -16406.574} C_VEL
LIN {X 0,Y 298.426,Z 369.309,A -85,B 0,C 180,E1 -16409.64,E2 -16409.64} C_VEL
LIN {X 0,Y 298.401,Z 369.313,A -85,B 0,C 180,E1 -16412.799,E2 -16412.799} C_VEL
LIN {X 0,Y 298.451,Z 369.307,A -85,B 0,C 180,E1 -16416.807,E2 -16416.807} C_VEL
LIN {X 0,Y 298.413,Z 369.31,A -85,B 0,C 180,E1 -16419.485,E2 -16419.485} C_VEL
LIN {X 0,Y 298.403,Z 369.311,A -85,B 0,C 180,E1 -16423.102,E2 -16423.102} C_VEL
LIN {X 0,Y 298.407,Z 369.312,A -85,B 0,C 180,E1 -16426.92,E2 -16426.92} C_VEL
LIN {X 0,Y 298.419,Z 369.309,A -85,B 0,C 180,E1 -16431.003,E2 -16431.003} C_VEL
LIN {X 0,Y 298.425,Z 369.312,A -85,B 0,C 180,E1 -16433.929,E2 -16433.929} C_VEL
LIN {X 0,Y 298.398,Z 369.316,A -85,B 0,C 180,E1 -16437.982,E2 -16437.982} C_VEL
LIN {X 0,Y 298.463,Z 369.307,A -85,B 0,C 180,E1 -16441.903,E2 -16441.903} C_VEL
LIN {X 0,Y 298.489,Z 369.301,A -85,B 0,C 180,E1 -16444.923,E2 -16444.923} C_VEL
LIN {X 0,Y 298.453,Z 369.305,A -85,B 0,C 180,E1 -16449.314,E2 -16449.314} C_VEL
LIN {X 0,Y 298.541,Z 369.299,A -85,B 0,C 180,E1 -16452.178,E2 -16452.178} C_VEL
LIN {X 0,Y 298.596,Z 369.287,A -85,B 0,C 180,E1 -16454.993,E2 -16454.993} C_VEL
LIN {X 0,Y 298.594,Z 369.288,A -85,B 0,C 180,E1 -16459.145,E2 -16459.145} C_VEL
LIN {X 0,Y 298.743,Z 369.273,A -85,B 0,C 180,E1 -16461.884,E2 -16461.884} C_VEL
LIN {X 0,Y 298.66,Z 369.28,A -85,B 0,C 180,E1 -16464.597,E2 -16464.597} C_VEL
LIN {X 0,Y 298.926,Z 369.247,A -85,B 0,C 180,E1 -16468.651,E2 -16468.651} C_VEL
LIN {X 0,Y 298.925,Z 369.247,A -85,B 0,C 180,E1 -16471.346,E2 -16471.346} C_VEL
LIN {X 0,Y 298.799,Z 369.262,A -85,B 0,C 180,E1 -16476.752,E2 -16476.752} C_VEL
LIN {X 0,Y 298.68,Z 369.279,A -85,B 0,C 180,E1 -16479.479,E2 -16479.479} C_VEL
LIN {X 0,Y 298.551,Z 369.295,A -85,B 0,C 180,E1 -16483.614,E2 -16483.614} C_VEL
LIN {X 0,Y 298.548,Z 369.295,A -85,B 0,C 180,E1 -16486.407,E2 -16486.407} C_VEL
LIN {X 0,Y 298.51,Z 369.302,A -85,B 0,C 180,E1 -16489.653,E2 -16489.653} C_VEL
LIN {X 0,Y 298.454,Z 369.308,A -85,B 0,C 180,E1 -16493.596,E2 -16493.596} C_VEL
LIN {X 0,Y 298.486,Z 369.302,A -85,B 0,C 180,E1 -16496.573,E2 -16496.573} C_VEL
LIN {X 0,Y 298.418,Z 369.313,A -85,B 0,C 180,E1 -16499.639,E2 -16499.639} C_VEL
LIN {X 0,Y 298.393,Z 369.313,A -85,B 0,C 180,E1 -16502.798,E2 -16502.798} C_VEL
LIN {X 0,Y 298.466,Z 369.304,A -85,B 0,C 180,E1 -16506.812,E2 -16506.812} C_VEL
LIN {X 0,Y 298.451,Z 369.306,A -85,B 0,C 180,E1 -16511.248,E2 -16511.248} C_VEL
LIN {X 0,Y 298.483,Z 369.302,A -85,B 0,C 180,E1 -16515.06,E2 -16515.06} C_VEL
LIN {X 0,Y 298.45,Z 369.305,A -85,B 0,C 180,E1 -16518.896,E2 -16518.896} C_VEL
LIN {X 0,Y 298.462,Z 369.306,A -85,B 0,C 180,E1 -16523.185,E2 -16523.185} C_VEL
LIN {X 0,Y 298.388,Z 369.314,A -85,B 0,C 180,E1 -16527.199,E2 -16527.199} C_VEL
LIN {X 0,Y 298.467,Z 369.307,A -85,B 0,C 180,E1 -16531.905,E2 -16531.905} C_VEL
LIN {X 0,Y 298.478,Z 369.302,A -85,B 0,C 180,E1 -16534.923,E2 -16534.923} C_VEL
LIN {X 0,Y 298.441,Z 369.31,A -85,B 0,C 180,E1 -16539.315,E2 -16539.315} C_VEL
LIN {X 0,Y 298.529,Z 369.297,A -85,B 0,C 180,E1 -16542.179,E2 -16542.179} C_VEL
LIN {X 0,Y 298.584,Z 369.289,A -85,B 0,C 180,E1 -16544.994,E2 -16544.994} C_VEL
LIN {X 0,Y 298.586,Z 369.291,A -85,B 0,C 180,E1 -16549.146,E2 -16549.146} C_VEL
LIN {X 0,Y 298.749,Z 369.27,A -85,B 0,C 180,E1 -16551.886,E2 -16551.886} C_VEL
LIN {X 0,Y 298.755,Z 369.267,A -85,B 0,C 180,E1 -16552.757,E2 -16552.757} C_VEL
LIN {X 0,Y 298.142,Z 369.348,A -85,B 0,C 180,E1 -16553.88,E2 -16553.88} C_VEL
LIN {X 0,Y 295.356,Z 369.698,A -85,B 0,C 180,E1 -16555.711,E2 -16555.711} C_VEL
LIN {X 0,Y 292.974,Z 369.994,A -85,B 0,C 180,E1 -16557.197,E2 -16557.197} C_VEL
LIN {X 0,Y 291.961,Z 370.116,A -85,B 0,C 180,E1 -16558.347,E2 -16558.347} C_VEL
LIN {X 0,Y 291.885,Z 370.123,A -85,B 0,C 180,E1 -16558.736,E2 -16558.736} C_VEL
LIN {X 0,Y 291.882,Z 370.128,A -85,B 0,C 180,E1 -16561.38,E2 -16561.38} C_VEL
LIN {X 0,Y 291.739,Z 370.143,A -85,B 0,C 180,E1 -16566.918,E2 -16566.918} C_VEL
LIN {X 0,Y 291.621,Z 370.159,A -85,B 0,C 180,E1 -16569.712,E2 -16569.712} C_VEL
LIN {X 0,Y 291.514,Z 370.171,A -85,B 0,C 180,E1 -16573.951,E2 -16573.951} C_VEL
LIN {X 0,Y 291.478,Z 370.175,A -85,B 0,C 180,E1 -16576.819,E2 -16576.819} C_VEL
LIN {X 0,Y 291.442,Z 370.179,A -85,B 0,C 180,E1 -16579.876,E2 -16579.876} C_VEL
LIN {X 0,Y 291.391,Z 370.185,A -85,B 0,C 180,E1 -16584.206,E2 -16584.206} C_VEL
LIN {X 0,Y 291.411,Z 370.187,A -85,B 0,C 180,E1 -16587.273,E2 -16587.273} C_VEL
LIN {X 0,Y 291.326,Z 370.193,A -85,B 0,C 180,E1 -16590.438,E2 -16590.438} C_VEL
LIN {X 0,Y 291.337,Z 370.194,A -85,B 0,C 180,E1 -16593.7,E2 -16593.7} C_VEL
LIN {X 0,Y 291.4,Z 370.188,A -85,B 0,C 180,E1 -16597.263,E2 -16597.263} C_VEL
LIN {X 0,Y 291.401,Z 370.185,A -85,B 0,C 180,E1 -16600.631,E2 -16600.631} C_VEL
LIN {X 0,Y 291.401,Z 370.184,A -85,B 0,C 180,E1 -16604.381,E2 -16604.381} C_VEL
LIN {X 0,Y 291.386,Z 370.186,A -85,B 0,C 180,E1 -16608.392,E2 -16608.392} C_VEL
LIN {X 0,Y 291.384,Z 370.191,A -85,B 0,C 180,E1 -16611.166,E2 -16611.166} C_VEL
LIN {X 0,Y 291.382,Z 370.186,A -85,B 0,C 180,E1 -16614.631,E2 -16614.631} C_VEL
LIN {X 0,Y 291.416,Z 370.244,A -85,B 0,C 180,E1 -16616.534,E2 -16616.534} C_VEL
LIN {X 0,Y 294.487,Z 385.285,A -85,B 0,C 180,E1 -16620.712,E2 -16620.712} C_VEL
LIN {X 0,Y 295.602,Z 391.5,A -85,B 0,C 180,E1 -16622.381,E2 -16622.381} C_VEL
LIN {X 0,Y 293.842,Z 406.131,A -85,B 0,C 180,E1 -16626.088,E2 -16626.088} C_VEL
LIN {X 0,Y 295.758,Z 432.701,A -85,B 0,C 180,E1 -16627.181,E2 -16627.181} C_VEL
LIN {X 0,Y 297.796,Z 453.438,A -85,B 0,C 180,E1 -16628.03,E2 -16628.03} C_VEL
LIN {X 0,Y 295.736,Z 516.456,A -85,B 0,C 180,E1 -16630.343,E2 -16630.343} C_VEL
LIN {X 0,Y 294.951,Z 529.231,A -85,B 0,C 180,E1 -16631.057,E2 -16631.057} C_VEL
LIN {X 0,Y 294.173,Z 540.485,A -85,B 0,C 180,E1 -16631.908,E2 -16631.908} C_VEL
LIN {X 0,Y 293.294,Z 552.752,A -85,B 0,C 180,E1 -16633.111,E2 -16633.111} C_VEL
LIN {X 0,Y 292.421,Z 563.77,A -85,B 0,C 180,E1 -16634.472,E2 -16634.472} C_VEL
LIN {X 0,Y 291.572,Z 574.154,A -85,B 0,C 180,E1 -16636.054,E2 -16636.054} C_VEL
LIN {X 0,Y 290.922,Z 583.439,A -85,B 0,C 180,E1 -16637.799,E2 -16637.799} C_VEL
LIN {X 0,Y 290.397,Z 592.493,A -85,B 0,C 180,E1 -16639.896,E2 -16639.896} C_VEL
LIN {X 0,Y 290.209,Z 599.665,A -85,B 0,C 180,E1 -16641.997,E2 -16641.997} C_VEL
LIN {X 0,Y 290.146,Z 604.551,A -85,B 0,C 180,E1 -16643.773,E2 -16643.773} C_VEL
LIN {X 0,Y 290.161,Z 608.995,A -85,B 0,C 180,E1 -16645.835,E2 -16645.835} C_VEL
LIN {X 0,Y 290.159,Z 611.309,A -85,B 0,C 180,E1 -16647.225,E2 -16647.225} C_VEL
LIN {X 0,Y 290.335,Z 613.155,A -85,B 0,C 180,E1 -16648.615,E2 -16648.615} C_VEL
LIN {X 0,Y 290.31,Z 614.435,A -85,B 0,C 180,E1 -16650.002,E2 -16650.002} C_VEL
LIN {X 0,Y 290.024,Z 615.232,A -85,B 0,C 180,E1 -16651.39,E2 -16651.39} C_VEL
LIN {X 0,Y 289.84,Z 615.608,A -85,B 0,C 180,E1 -16652.781,E2 -16652.781} C_VEL
LIN {X 0,Y 289.707,Z 615.537,A -85,B 0,C 180,E1 -16654.175,E2 -16654.175} C_VEL
LIN {X 0,Y 289.676,Z 614.824,A -85,B 0,C 180,E1 -16655.885,E2 -16655.885} C_VEL
LIN {X 0,Y 289.816,Z 612.689,A -85,B 0,C 180,E1 -16658.368,E2 -16658.368} C_VEL
LIN {X 0,Y 290.27,Z 609.81,A -85,B 0,C 180,E1 -16660.464,E2 -16660.464} C_VEL
LIN {X 0,Y 291.079,Z 605.932,A -85,B 0,C 180,E1 -16662.552,E2 -16662.552} C_VEL
LIN {X 0,Y 292.451,Z 600.97,A -85,B 0,C 180,E1 -16664.617,E2 -16664.617} C_VEL
LIN {X 0,Y 293.953,Z 594.832,A -85,B 0,C 180,E1 -16666.674,E2 -16666.674} C_VEL
LIN {X 0,Y 296.226,Z 587.35,A -85,B 0,C 180,E1 -16668.682,E2 -16668.682} C_VEL
LIN {X 0,Y 298.903,Z 578.211,A -85,B 0,C 180,E1 -16670.653,E2 -16670.653} C_VEL
LIN {X 0,Y 302.078,Z 567.091,A -85,B 0,C 180,E1 -16672.576,E2 -16672.576} C_VEL
LIN {X 0,Y 305.143,Z 555.681,A -85,B 0,C 180,E1 -16674.132,E2 -16674.132} C_VEL
LIN {X 0,Y 307.82,Z 544.743,A -85,B 0,C 180,E1 -16675.348,E2 -16675.348} C_VEL
LIN {X 0,Y 310.565,Z 532.988,A -85,B 0,C 180,E1 -16676.368,E2 -16676.368} C_VEL
LIN {X 0,Y 313.478,Z 518.003,A -85,B 0,C 180,E1 -16677.363,E2 -16677.363} C_VEL
LIN {X 0,Y 315.655,Z 501.972,A -85,B 0,C 180,E1 -16678.148,E2 -16678.148} C_VEL
LIN {X 0,Y 320.397,Z 459.004,A -85,B 0,C 180,E1 -16679.888,E2 -16679.888} C_VEL
LIN {X 0,Y 320.336,Z 449.291,A -85,B 0,C 180,E1 -16680.569,E2 -16680.569} C_VEL
LIN {X 0,Y 319.479,Z 436.698,A -85,B 0,C 180,E1 -16681.702,E2 -16681.702} C_VEL
LIN {X 0,Y 318.264,Z 425.685,A -85,B 0,C 180,E1 -16682.915,E2 -16682.915} C_VEL
LIN {X 0,Y 316.736,Z 421.717,A -85,B 0,C 180,E1 -16683.731,E2 -16683.731} C_VEL
LIN {X 0,Y 314.506,Z 416.421,A -85,B 0,C 180,E1 -16685,E2 -16685} C_VEL
LIN {X 0,Y 311.865,Z 410.412,A -85,B 0,C 180,E1 -16686.732,E2 -16686.732} C_VEL
LIN {X 0,Y 308.157,Z 402.631,A -85,B 0,C 180,E1 -16689.945,E2 -16689.945} C_VEL
LIN {X 0,Y 306.118,Z 398.947,A -85,B 0,C 180,E1 -16692.824,E2 -16692.824} C_VEL
LIN {X 0,Y 305.587,Z 397.072,A -85,B 0,C 180,E1 -16695.258,E2 -16695.258} C_VEL
LIN {X 0,Y 305.954,Z 396.325,A -85,B 0,C 180,E1 -16697.315,E2 -16697.315} C_VEL
LIN {X 0,Y 306.872,Z 396.407,A -85,B 0,C 180,E1 -16699.094,E2 -16699.094} C_VEL
LIN {X 0,Y 309.856,Z 399.049,A -85,B 0,C 180,E1 -16702.355,E2 -16702.355} C_VEL
LIN {X 0,Y 313.384,Z 403.323,A -85,B 0,C 180,E1 -16704.865,E2 -16704.865} C_VEL
LIN {X 0,Y 316.378,Z 407.389,A -85,B 0,C 180,E1 -16706.542,E2 -16706.542} C_VEL
LIN {X 0,Y 319.361,Z 411.733,A -85,B 0,C 180,E1 -16707.972,E2 -16707.972} C_VEL
LIN {X 0,Y 323.28,Z 418.315,A -85,B 0,C 180,E1 -16709.646,E2 -16709.646} C_VEL
LIN {X 0,Y 324.032,Z 419.822,A -85,B 0,C 180,E1 -16709.958,E2 -16709.958} C_VEL
LIN {X 0,Y 316.941,Z 479.208,A -85,B 0,C 180,E1 -16712.426,E2 -16712.426} C_VEL
LIN {X 0,Y 315.191,Z 492.708,A -85,B 0,C 180,E1 -16713.248,E2 -16713.248} C_VEL
LIN {X 0,Y 313.097,Z 505.329,A -85,B 0,C 180,E1 -16714.268,E2 -16714.268} C_VEL
LIN {X 0,Y 310.723,Z 516.945,A -85,B 0,C 180,E1 -16715.469,E2 -16715.469} C_VEL
LIN {X 0,Y 308.255,Z 527.576,A -85,B 0,C 180,E1 -16716.841,E2 -16716.841} C_VEL
LIN {X 0,Y 305.05,Z 539.203,A -85,B 0,C 180,E1 -16718.724,E2 -16718.724} C_VEL
LIN {X 0,Y 302.213,Z 548.443,A -85,B 0,C 180,E1 -16720.647,E2 -16720.647} C_VEL
LIN {X 0,Y 299.733,Z 555.932,A -85,B 0,C 180,E1 -16722.605,E2 -16722.605} C_VEL
LIN {X 0,Y 297.892,Z 561.041,A -85,B 0,C 180,E1 -16724.257,E2 -16724.257} C_VEL
LIN {X 0,Y 295.97,Z 566.005,A -85,B 0,C 180,E1 -16726.263,E2 -16726.263} C_VEL
LIN {X 0,Y 294.498,Z 569.486,A -85,B 0,C 180,E1 -16728.085,E2 -16728.085} C_VEL
LIN {X 0,Y 292.855,Z 572.623,A -85,B 0,C 180,E1 -16730.329,E2 -16730.329} C_VEL
LIN {X 0,Y 292.158,Z 573.923,A -85,B 0,C 180,E1 -16731.701,E2 -16731.701} C_VEL
LIN {X 0,Y 291.58,Z 574.755,A -85,B 0,C 180,E1 -16733.078,E2 -16733.078} C_VEL
LIN {X 0,Y 291.243,Z 575.171,A -85,B 0,C 180,E1 -16734.461,E2 -16734.461} C_VEL
LIN {X 0,Y 290.885,Z 575.197,A -85,B 0,C 180,E1 -16735.843,E2 -16735.843} C_VEL
LIN {X 0,Y 290.456,Z 574.797,A -85,B 0,C 180,E1 -16737.226,E2 -16737.226} C_VEL
LIN {X 0,Y 290.161,Z 573.943,A -85,B 0,C 180,E1 -16738.612,E2 -16738.612} C_VEL
LIN {X 0,Y 290.009,Z 572.673,A -85,B 0,C 180,E1 -16740,E2 -16740} C_VEL
LIN {X 0,Y 289.902,Z 569.928,A -85,B 0,C 180,E1 -16742.084,E2 -16742.084} C_VEL
LIN {X 0,Y 290.07,Z 566.121,A -85,B 0,C 180,E1 -16744.168,E2 -16744.168} C_VEL
LIN {X 0,Y 290.214,Z 560.652,A -85,B 0,C 180,E1 -16746.443,E2 -16746.443} C_VEL
LIN {X 0,Y 290.633,Z 553.647,A -85,B 0,C 180,E1 -16748.693,E2 -16748.693} C_VEL
LIN {X 0,Y 291.207,Z 545.542,A -85,B 0,C 180,E1 -16750.78,E2 -16750.78} C_VEL
LIN {X 0,Y 291.826,Z 537.27,A -85,B 0,C 180,E1 -16752.518,E2 -16752.518} C_VEL
LIN {X 0,Y 292.698,Z 526.104,A -85,B 0,C 180,E1 -16754.425,E2 -16754.425} C_VEL
LIN {X 0,Y 293.651,Z 514.82,A -85,B 0,C 180,E1 -16755.976,E2 -16755.976} C_VEL
LIN {X 0,Y 294.388,Z 502.238,A -85,B 0,C 180,E1 -16757.357,E2 -16757.357} C_VEL
LIN {X 0,Y 295.153,Z 488.943,A -85,B 0,C 180,E1 -16758.481,E2 -16758.481} C_VEL
LIN {X 0,Y 295.783,Z 475.157,A -85,B 0,C 180,E1 -16759.339,E2 -16759.339} C_VEL
LIN {X 0,Y 296.379,Z 458.364,A -85,B 0,C 180,E1 -16760.02,E2 -16760.02} C_VEL
LIN {X 0,Y 298.576,Z 393.167,A -85,B 0,C 180,E1 -16762.34,E2 -16762.34} C_VEL
LIN {X 0,Y 291.433,Z 370.177,A -85,B 0,C 180,E1 -16763.528,E2 -16763.528} C_VEL
LIN {X 0,Y 291.428,Z 370.181,A -85,B 0,C 180,E1 -16767.271,E2 -16767.271} C_VEL
LIN {X 0,Y 291.343,Z 370.195,A -85,B 0,C 180,E1 -16770.436,E2 -16770.436} C_VEL
LIN {X 0,Y 291.35,Z 370.19,A -85,B 0,C 180,E1 -16773.698,E2 -16773.698} C_VEL
LIN {X 0,Y 291.386,Z 370.186,A -85,B 0,C 180,E1 -16777.254,E2 -16777.254} C_VEL
LIN {X 0,Y 291.339,Z 370.193,A -85,B 0,C 180,E1 -16780.641,E2 -16780.641} C_VEL
LIN {X 0,Y 291.295,Z 370.201,A -85,B 0,C 180,E1 -16784.401,E2 -16784.401} C_VEL
LIN {X 0,Y 291.331,Z 370.196,A -85,B 0,C 180,E1 -16788.403,E2 -16788.403} C_VEL
LIN {X 0,Y 291.368,Z 370.187,A -85,B 0,C 180,E1 -16791.159,E2 -16791.159} C_VEL
LIN {X 0,Y 291.366,Z 370.19,A -85,B 0,C 180,E1 -16794.625,E2 -16794.625} C_VEL
LIN {X 0,Y 291.375,Z 370.19,A -85,B 0,C 180,E1 -16797.95,E2 -16797.95} C_VEL
LIN {X 0,Y 291.381,Z 370.186,A -85,B 0,C 180,E1 -16801.157,E2 -16801.157} C_VEL
LIN {X 0,Y 291.418,Z 370.186,A -85,B 0,C 180,E1 -16804.271,E2 -16804.271} C_VEL
LIN {X 0,Y 291.385,Z 370.185,A -85,B 0,C 180,E1 -16807.298,E2 -16807.298} C_VEL
LIN {X 0,Y 291.462,Z 370.18,A -85,B 0,C 180,E1 -16810.269,E2 -16810.269} C_VEL
LIN {X 0,Y 291.558,Z 370.165,A -85,B 0,C 180,E1 -16814.622,E2 -16814.622} C_VEL
LIN {X 0,Y 291.538,Z 370.167,A -85,B 0,C 180,E1 -16818.879,E2 -16818.879} C_VEL
LIN {X 0,Y 291.69,Z 370.15,A -85,B 0,C 180,E1 -16821.686,E2 -16821.686} C_VEL
LIN {X 0,Y 291.63,Z 370.156,A -85,B 0,C 180,E1 -16824.467,E2 -16824.467} C_VEL
LIN {X 0,Y 291.892,Z 370.124,A -85,B 0,C 180,E1 -16828.619,E2 -16828.619} C_VEL
LIN {X 0,Y 291.891,Z 370.124,A -85,B 0,C 180,E1 -16831.378,E2 -16831.378} C_VEL
LIN {X 0,Y 291.747,Z 370.141,A -85,B 0,C 180,E1 -16836.916,E2 -16836.916} C_VEL
LIN {X 0,Y 291.629,Z 370.159,A -85,B 0,C 180,E1 -16839.71,E2 -16839.71} C_VEL
LIN {X 0,Y 291.521,Z 370.173,A -85,B 0,C 180,E1 -16843.949,E2 -16843.949} C_VEL
LIN {X 0,Y 291.486,Z 370.173,A -85,B 0,C 180,E1 -16846.816,E2 -16846.816} C_VEL
LIN {X 0,Y 291.448,Z 370.183,A -85,B 0,C 180,E1 -16849.873,E2 -16849.873} C_VEL
LIN {X 0,Y 291.397,Z 370.187,A -85,B 0,C 180,E1 -16854.204,E2 -16854.204} C_VEL
LIN {X 0,Y 291.419,Z 370.183,A -85,B 0,C 180,E1 -16857.27,E2 -16857.27} C_VEL
LIN {X 0,Y 291.335,Z 370.192,A -85,B 0,C 180,E1 -16860.435,E2 -16860.435} C_VEL
LIN {X 0,Y 291.341,Z 370.195,A -85,B 0,C 180,E1 -16863.697,E2 -16863.697} C_VEL
LIN {X 0,Y 291.4,Z 370.185,A -85,B 0,C 180,E1 -16867.26,E2 -16867.26} C_VEL
LIN {X 0,Y 291.401,Z 370.183,A -85,B 0,C 180,E1 -16870.629,E2 -16870.629} C_VEL
LIN {X 0,Y 291.401,Z 370.185,A -85,B 0,C 180,E1 -16874.378,E2 -16874.378} C_VEL
LIN {X 0,Y 291.384,Z 370.186,A -85,B 0,C 180,E1 -16878.389,E2 -16878.389} C_VEL
LIN {X 0,Y 291.381,Z 370.187,A -85,B 0,C 180,E1 -16881.163,E2 -16881.163} C_VEL
LIN {X 0,Y 291.378,Z 370.187,A -85,B 0,C 180,E1 -16884.629,E2 -16884.629} C_VEL
LIN {X 0,Y 291.364,Z 370.191,A -85,B 0,C 180,E1 -16887.95,E2 -16887.95} C_VEL
LIN {X 0,Y 291.381,Z 370.188,A -85,B 0,C 180,E1 -16891.158,E2 -16891.158} C_VEL
LIN {X 0,Y 291.413,Z 370.183,A -85,B 0,C 180,E1 -16894.272,E2 -16894.272} C_VEL
LIN {X 0,Y 291.373,Z 370.189,A -85,B 0,C 180,E1 -16897.299,E2 -16897.299} C_VEL
LIN {X 0,Y 291.449,Z 370.179,A -85,B 0,C 180,E1 -16900.27,E2 -16900.27} C_VEL
LIN {X 0,Y 291.546,Z 370.165,A -85,B 0,C 180,E1 -16904.623,E2 -16904.623} C_VEL
LIN {X 0,Y 291.529,Z 370.168,A -85,B 0,C 180,E1 -16908.88,E2 -16908.88} C_VEL
LIN {X 0,Y 291.7,Z 370.15,A -85,B 0,C 180,E1 -16911.688,E2 -16911.688} C_VEL
LIN {X 0,Y 291.623,Z 370.156,A -85,B 0,C 180,E1 -16914.468,E2 -16914.468} C_VEL
LIN {X 0,Y 291.885,Z 370.123,A -85,B 0,C 180,E1 -16918.736,E2 -16918.736} C_VEL
LIN {X 0,Y 291.192,Z 370.212,A -85,B 0,C 180,E1 -16919.888,E2 -16919.888} C_VEL
LIN {X 0,Y 288.18,Z 370.587,A -85,B 0,C 180,E1 -16921.759,E2 -16921.759} C_VEL
LIN {X 0,Y 285.642,Z 370.903,A -85,B 0,C 180,E1 -16923.279,E2 -16923.279} C_VEL
LIN {X 0,Y 284.588,Z 371.032,A -85,B 0,C 180,E1 -16924.461,E2 -16924.461} C_VEL
LIN {X 0,Y 284.522,Z 371.04,A -85,B 0,C 180,E1 -16924.862,E2 -16924.862} C_VEL
LIN {X 0,Y 284.691,Z 371.022,A -85,B 0,C 180,E1 -16927.09,E2 -16927.09} C_VEL
LIN {X 0,Y 284.558,Z 371.037,A -85,B 0,C 180,E1 -16929.956,E2 -16929.956} C_VEL
LIN {X 0,Y 284.474,Z 371.047,A -85,B 0,C 180,E1 -16934.303,E2 -16934.303} C_VEL
LIN {X 0,Y 284.417,Z 371.058,A -85,B 0,C 180,E1 -16937.249,E2 -16937.249} C_VEL
LIN {X 0,Y 284.37,Z 371.059,A -85,B 0,C 180,E1 -16940.243,E2 -16940.243} C_VEL
LIN {X 0,Y 284.361,Z 371.062,A -85,B 0,C 180,E1 -16943.876,E2 -16943.876} C_VEL
LIN {X 0,Y 284.386,Z 371.061,A -85,B 0,C 180,E1 -16947.174,E2 -16947.174} C_VEL
LIN {X 0,Y 284.286,Z 371.075,A -85,B 0,C 180,E1 -16951.276,E2 -16951.276} C_VEL
LIN {X 0,Y 284.356,Z 371.066,A -85,B 0,C 180,E1 -16955.356,E2 -16955.356} C_VEL
LIN {X 0,Y 284.332,Z 371.064,A -85,B 0,C 180,E1 -16958.166,E2 -16958.166} C_VEL
LIN {X 0,Y 284.339,Z 371.064,A -85,B 0,C 180,E1 -16962.143,E2 -16962.143} C_VEL
LIN {X 0,Y 284.348,Z 371.061,A -85,B 0,C 180,E1 -16966.21,E2 -16966.21} C_VEL
LIN {X 0,Y 284.347,Z 371.063,A -85,B 0,C 180,E1 -16970.015,E2 -16970.015} C_VEL
LIN {X 0,Y 284.351,Z 371.063,A -85,B 0,C 180,E1 -16973.619,E2 -16973.619} C_VEL
LIN {X 0,Y 284.399,Z 371.121,A -85,B 0,C 180,E1 -16976.339,E2 -16976.339} C_VEL
LIN {X 0,Y 287.503,Z 386.555,A -85,B 0,C 180,E1 -16980.734,E2 -16980.734} C_VEL
LIN {X 0,Y 288.394,Z 390.98,A -85,B 0,C 180,E1 -16981.958,E2 -16981.958} C_VEL
LIN {X 0,Y 288.176,Z 395.641,A -85,B 0,C 180,E1 -16983.183,E2 -16983.183} C_VEL
LIN {X 0,Y 286.864,Z 406.063,A -85,B 0,C 180,E1 -16985.822,E2 -16985.822} C_VEL
LIN {X 0,Y 288.624,Z 432.016,A -85,B 0,C 180,E1 -16986.899,E2 -16986.899} C_VEL
LIN {X 0,Y 290.798,Z 453.531,A -85,B 0,C 180,E1 -16987.81,E2 -16987.81} C_VEL
LIN {X 0,Y 288.666,Z 516.52,A -85,B 0,C 180,E1 -16990.212,E2 -16990.212} C_VEL
LIN {X 0,Y 287.891,Z 529.091,A -85,B 0,C 180,E1 -16990.945,E2 -16990.945} C_VEL
LIN {X 0,Y 286.943,Z 542.088,A -85,B 0,C 180,E1 -16991.99,E2 -16991.99} C_VEL
LIN {X 0,Y 286.14,Z 553.53,A -85,B 0,C 180,E1 -16993.183,E2 -16993.183} C_VEL
LIN {X 0,Y 285.198,Z 564.733,A -85,B 0,C 180,E1 -16994.64,E2 -16994.64} C_VEL
LIN {X 0,Y 284.366,Z 575.661,A -85,B 0,C 180,E1 -16996.423,E2 -16996.423} C_VEL
LIN {X 0,Y 283.777,Z 584.611,A -85,B 0,C 180,E1 -16998.212,E2 -16998.212} C_VEL
LIN {X 0,Y 283.298,Z 593.259,A -85,B 0,C 180,E1 -17000.362,E2 -17000.362} C_VEL
LIN {X 0,Y 283.141,Z 600.17,A -85,B 0,C 180,E1 -17002.514,E2 -17002.514} C_VEL
LIN {X 0,Y 283.1,Z 604.748,A -85,B 0,C 180,E1 -17004.303,E2 -17004.303} C_VEL
LIN {X 0,Y 283.15,Z 609.035,A -85,B 0,C 180,E1 -17006.444,E2 -17006.444} C_VEL
LIN {X 0,Y 283.292,Z 612.114,A -85,B 0,C 180,E1 -17008.58,E2 -17008.58} C_VEL
LIN {X 0,Y 283.265,Z 613.544,A -85,B 0,C 180,E1 -17010.002,E2 -17010.002} C_VEL
LIN {X 0,Y 282.963,Z 614.426,A -85,B 0,C 180,E1 -17011.425,E2 -17011.425} C_VEL
LIN {X 0,Y 282.778,Z 614.879,A -85,B 0,C 180,E1 -17012.851,E2 -17012.851} C_VEL
LIN {X 0,Y 282.636,Z 614.907,A -85,B 0,C 180,E1 -17014.28,E2 -17014.28} C_VEL
LIN {X 0,Y 282.604,Z 614.433,A -85,B 0,C 180,E1 -17015.871,E2 -17015.871} C_VEL
LIN {X 0,Y 282.756,Z 612.38,A -85,B 0,C 180,E1 -17018.578,E2 -17018.578} C_VEL
LIN {X 0,Y 283.241,Z 609.692,A -85,B 0,C 180,E1 -17020.727,E2 -17020.727} C_VEL
LIN {X 0,Y 284.137,Z 606.018,A -85,B 0,C 180,E1 -17022.864,E2 -17022.864} C_VEL
LIN {X 0,Y 285.568,Z 601.278,A -85,B 0,C 180,E1 -17024.977,E2 -17024.977} C_VEL
LIN {X 0,Y 287.485,Z 594.472,A -85,B 0,C 180,E1 -17027.368,E2 -17027.368} C_VEL
LIN {X 0,Y 289.974,Z 586.888,A -85,B 0,C 180,E1 -17029.468,E2 -17029.468} C_VEL
LIN {X 0,Y 292.921,Z 577.869,A -85,B 0,C 180,E1 -17031.464,E2 -17031.464} C_VEL
LIN {X 0,Y 296.276,Z 566.905,A -85,B 0,C 180,E1 -17033.413,E2 -17033.413} C_VEL
LIN {X 0,Y 299.532,Z 555.731,A -85,B 0,C 180,E1 -17034.984,E2 -17034.984} C_VEL
LIN {X 0,Y 302.392,Z 545.012,A -85,B 0,C 180,E1 -17036.207,E2 -17036.207} C_VEL
LIN {X 0,Y 305.705,Z 531.794,A -85,B 0,C 180,E1 -17037.375,E2 -17037.375} C_VEL
LIN {X 0,Y 308.526,Z 518.083,A -85,B 0,C 180,E1 -17038.302,E2 -17038.302} C_VEL
LIN {X 0,Y 310.837,Z 502.825,A -85,B 0,C 180,E1 -17039.087,E2 -17039.087} C_VEL
LIN {X 0,Y 315.944,Z 460.252,A -85,B 0,C 180,E1 -17040.853,E2 -17040.853} C_VEL
LIN {X 0,Y 315.933,Z 450,A -85,B 0,C 180,E1 -17041.625,E2 -17041.625} C_VEL
LIN {X 0,Y 315.198,Z 437.155,A -85,B 0,C 180,E1 -17042.866,E2 -17042.866} C_VEL
LIN {X 0,Y 314.45,Z 429.853,A -85,B 0,C 180,E1 -17043.735,E2 -17043.735} C_VEL
LIN {X 0,Y 313.064,Z 426.15,A -85,B 0,C 180,E1 -17044.554,E2 -17044.554} C_VEL
LIN {X 0,Y 311.397,Z 421.898,A -85,B 0,C 180,E1 -17045.619,E2 -17045.619} C_VEL
LIN {X 0,Y 309.129,Z 416.279,A -85,B 0,C 180,E1 -17047.276,E2 -17047.276} C_VEL
LIN {X 0,Y 305.949,Z 409.06,A -85,B 0,C 180,E1 -17050.349,E2 -17050.349} C_VEL
LIN {X 0,Y 304.17,Z 405.481,A -85,B 0,C 180,E1 -17053.25,E2 -17053.25} C_VEL
LIN {X 0,Y 303.817,Z 403.774,A -85,B 0,C 180,E1 -17055.585,E2 -17055.585} C_VEL
LIN {X 0,Y 304.478,Z 403.117,A -85,B 0,C 180,E1 -17057.98,E2 -17057.98} C_VEL
LIN {X 0,Y 305.283,Z 403.582,A -85,B 0,C 180,E1 -17059.44,E2 -17059.44} C_VEL
LIN {X 0,Y 308.199,Z 406.249,A -85,B 0,C 180,E1 -17062.505,E2 -17062.505} C_VEL
LIN {X 0,Y 311.162,Z 410.11,A -85,B 0,C 180,E1 -17064.686,E2 -17064.686} C_VEL
LIN {X 0,Y 313.853,Z 413.881,A -85,B 0,C 180,E1 -17066.258,E2 -17066.258} C_VEL
LIN {X 0,Y 316.959,Z 418.575,A -85,B 0,C 180,E1 -17067.814,E2 -17067.814} C_VEL
LIN {X 0,Y 319.626,Z 423.415,A -85,B 0,C 180,E1 -17069.043,E2 -17069.043} C_VEL
LIN {X 0,Y 312.311,Z 480.2,A -85,B 0,C 180,E1 -17071.462,E2 -17071.462} C_VEL
LIN {X 0,Y 310.484,Z 493.251,A -85,B 0,C 180,E1 -17072.271,E2 -17072.271} C_VEL
LIN {X 0,Y 308.249,Z 505.776,A -85,B 0,C 180,E1 -17073.295,E2 -17073.295} C_VEL
LIN {X 0,Y 305.481,Z 518.4,A -85,B 0,C 180,E1 -17074.628,E2 -17074.628} C_VEL
LIN {X 0,Y 302.5,Z 530.001,A -85,B 0,C 180,E1 -17076.192,E2 -17076.192} C_VEL
LIN {X 0,Y 299.384,Z 540.401,A -85,B 0,C 180,E1 -17077.938,E2 -17077.938} C_VEL
LIN {X 0,Y 296.341,Z 549.502,A -85,B 0,C 180,E1 -17079.886,E2 -17079.886} C_VEL
LIN {X 0,Y 293.636,Z 556.913,A -85,B 0,C 180,E1 -17081.871,E2 -17081.871} C_VEL
LIN {X 0,Y 291.294,Z 562.868,A -85,B 0,C 180,E1 -17083.891,E2 -17083.891} C_VEL
LIN {X 0,Y 289.247,Z 567.566,A -85,B 0,C 180,E1 -17085.938,E2 -17085.938} C_VEL
LIN {X 0,Y 287.881,Z 570.462,A -85,B 0,C 180,E1 -17087.563,E2 -17087.563} C_VEL
LIN {X 0,Y 285.964,Z 573.745,A -85,B 0,C 180,E1 -17090.094,E2 -17090.094} C_VEL
LIN {X 0,Y 285.214,Z 574.877,A -85,B 0,C 180,E1 -17091.498,E2 -17091.498} C_VEL
LIN {X 0,Y 284.599,Z 575.604,A -85,B 0,C 180,E1 -17092.907,E2 -17092.907} C_VEL
LIN {X 0,Y 284.218,Z 575.921,A -85,B 0,C 180,E1 -17094.323,E2 -17094.323} C_VEL
LIN {X 0,Y 283.842,Z 575.802,A -85,B 0,C 180,E1 -17095.74,E2 -17095.74} C_VEL
LIN {X 0,Y 283.406,Z 575.263,A -85,B 0,C 180,E1 -17097.157,E2 -17097.157} C_VEL
LIN {X 0,Y 283.088,Z 574.313,A -85,B 0,C 180,E1 -17098.577,E2 -17098.577} C_VEL
LIN {X 0,Y 282.913,Z 572.937,A -85,B 0,C 180,E1 -17100,E2 -17100} C_VEL
LIN {X 0,Y 282.812,Z 570.01,A -85,B 0,C 180,E1 -17102.136,E2 -17102.136} C_VEL
LIN {X 0,Y 283.002,Z 566.003,A -85,B 0,C 180,E1 -17104.272,E2 -17104.272} C_VEL
LIN {X 0,Y 283.108,Z 560.881,A -85,B 0,C 180,E1 -17106.383,E2 -17106.383} C_VEL
LIN {X 0,Y 283.533,Z 554.251,A -85,B 0,C 180,E1 -17108.553,E2 -17108.553} C_VEL
LIN {X 0,Y 284.084,Z 546.133,A -85,B 0,C 180,E1 -17110.693,E2 -17110.693} C_VEL
LIN {X 0,Y 284.7,Z 537.87,A -85,B 0,C 180,E1 -17112.474,E2 -17112.474} C_VEL
LIN {X 0,Y 285.604,Z 526.73,A -85,B 0,C 180,E1 -17114.427,E2 -17114.427} C_VEL
LIN {X 0,Y 286.504,Z 515.47,A -85,B 0,C 180,E1 -17116.019,E2 -17116.019} C_VEL
LIN {X 0,Y 287.298,Z 502.892,A -85,B 0,C 180,E1 -17117.435,E2 -17117.435} C_VEL
LIN {X 0,Y 288.072,Z 489.696,A -85,B 0,C 180,E1 -17118.583,E2 -17118.583} C_VEL
LIN {X 0,Y 288.702,Z 476.064,A -85,B 0,C 180,E1 -17119.463,E2 -17119.463} C_VEL
LIN {X 0,Y 289.291,Z 459.711,A -85,B 0,C 180,E1 -17120.162,E2 -17120.162} C_VEL
LIN {X 0,Y 291.507,Z 394.204,A -85,B 0,C 180,E1 -17122.583,E2 -17122.583} C_VEL
LIN {X 0,Y 284.42,Z 371.119,A -85,B 0,C 180,E1 -17123.776,E2 -17123.776} C_VEL
LIN {X 0,Y 284.338,Z 371.066,A -85,B 0,C 180,E1 -17128.01,E2 -17128.01} C_VEL
LIN {X 0,Y 284.301,Z 371.068,A -85,B 0,C 180,E1 -17131.274,E2 -17131.274} C_VEL
LIN {X 0,Y 284.346,Z 371.063,A -85,B 0,C 180,E1 -17135.347,E2 -17135.347} C_VEL
LIN {X 0,Y 284.324,Z 371.07,A -85,B 0,C 180,E1 -17138.167,E2 -17138.167} C_VEL
LIN {X 0,Y 284.274,Z 371.074,A -85,B 0,C 180,E1 -17142.124,E2 -17142.124} C_VEL
LIN {X 0,Y 284.26,Z 371.078,A -85,B 0,C 180,E1 -17146.188,E2 -17146.188} C_VEL
LIN {X 0,Y 284.311,Z 371.07,A -85,B 0,C 180,E1 -17150.023,E2 -17150.023} C_VEL
LIN {X 0,Y 284.341,Z 371.064,A -85,B 0,C 180,E1 -17153.614,E2 -17153.614} C_VEL
LIN {X 0,Y 284.312,Z 371.067,A -85,B 0,C 180,E1 -17157.188,E2 -17157.188} C_VEL
LIN {X 0,Y 284.359,Z 371.064,A -85,B 0,C 180,E1 -17160.374,E2 -17160.374} C_VEL
LIN {X 0,Y 284.38,Z 371.06,A -85,B 0,C 180,E1 -17163.585,E2 -17163.585} C_VEL
LIN {X 0,Y 284.37,Z 371.06,A -85,B 0,C 180,E1 -17166.706,E2 -17166.706} C_VEL
LIN {X 0,Y 284.407,Z 371.055,A -85,B 0,C 180,E1 -17171.26,E2 -17171.26} C_VEL
LIN {X 0,Y 284.495,Z 371.046,A -85,B 0,C 180,E1 -17174.458,E2 -17174.458} C_VEL
LIN {X 0,Y 284.49,Z 371.046,A -85,B 0,C 180,E1 -17178.6,E2 -17178.6} C_VEL
LIN {X 0,Y 284.641,Z 371.027,A -85,B 0,C 180,E1 -17181.479,E2 -17181.479} C_VEL
LIN {X 0,Y 284.6,Z 371.033,A -85,B 0,C 180,E1 -17184.33,E2 -17184.33} C_VEL
LIN {X 0,Y 284.858,Z 371,A -85,B 0,C 180,E1 -17188.585,E2 -17188.585} C_VEL
LIN {X 0,Y 284.857,Z 371,A -85,B 0,C 180,E1 -17191.412,E2 -17191.412} C_VEL
LIN {X 0,Y 284.699,Z 371.019,A -85,B 0,C 180,E1 -17197.088,E2 -17197.088} C_VEL
LIN {X 0,Y 284.566,Z 371.04,A -85,B 0,C 180,E1 -17199.954,E2 -17199.954} C_VEL
LIN {X 0,Y 284.481,Z 371.048,A -85,B 0,C 180,E1 -17204.301,E2 -17204.301} C_VEL
LIN {X 0,Y 284.424,Z 371.054,A -85,B 0,C 180,E1 -17207.247,E2 -17207.247} C_VEL
LIN {X 0,Y 284.376,Z 371.06,A -85,B 0,C 180,E1 -17210.24,E2 -17210.24} C_VEL
LIN {X 0,Y 284.367,Z 371.065,A -85,B 0,C 180,E1 -17213.874,E2 -17213.874} C_VEL
LIN {X 0,Y 284.394,Z 371.057,A -85,B 0,C 180,E1 -17217.172,E2 -17217.172} C_VEL
LIN {X 0,Y 284.294,Z 371.069,A -85,B 0,C 180,E1 -17221.272,E2 -17221.272} C_VEL
LIN {X 0,Y 284.357,Z 371.063,A -85,B 0,C 180,E1 -17225.353,E2 -17225.353} C_VEL
LIN {X 0,Y 284.332,Z 371.066,A -85,B 0,C 180,E1 -17228.163,E2 -17228.163} C_VEL
LIN {X 0,Y 284.339,Z 371.066,A -85,B 0,C 180,E1 -17232.14,E2 -17232.14} C_VEL
LIN {X 0,Y 284.347,Z 371.064,A -85,B 0,C 180,E1 -17236.207,E2 -17236.207} C_VEL
LIN {X 0,Y 284.344,Z 371.065,A -85,B 0,C 180,E1 -17240.012,E2 -17240.012} C_VEL
LIN {X 0,Y 284.347,Z 371.067,A -85,B 0,C 180,E1 -17243.616,E2 -17243.616} C_VEL
LIN {X 0,Y 284.3,Z 371.069,A -85,B 0,C 180,E1 -17247.188,E2 -17247.188} C_VEL
LIN {X 0,Y 284.353,Z 371.062,A -85,B 0,C 180,E1 -17250.376,E2 -17250.376} C_VEL
LIN {X 0,Y 284.373,Z 371.064,A -85,B 0,C 180,E1 -17253.586,E2 -17253.586} C_VEL
LIN {X 0,Y 284.358,Z 371.06,A -85,B 0,C 180,E1 -17256.706,E2 -17256.706} C_VEL
LIN {X 0,Y 284.395,Z 371.059,A -85,B 0,C 180,E1 -17261.261,E2 -17261.261} C_VEL
LIN {X 0,Y 284.483,Z 371.044,A -85,B 0,C 180,E1 -17264.459,E2 -17264.459} C_VEL
LIN {X 0,Y 284.481,Z 371.046,A -85,B 0,C 180,E1 -17268.601,E2 -17268.601} C_VEL
LIN {X 0,Y 284.65,Z 371.029,A -85,B 0,C 180,E1 -17271.481,E2 -17271.481} C_VEL
LIN {X 0,Y 284.593,Z 371.031,A -85,B 0,C 180,E1 -17274.331,E2 -17274.331} C_VEL
LIN {X 0,Y 284.85,Z 370.999,A -85,B 0,C 180,E1 -17278.738,E2 -17278.738} C_VEL
LIN {X 0,Y 284.848,Z 371.004,A -85,B 0,C 180,E1 -17281.414,E2 -17281.414} C_VEL
LIN {X 0,Y 284.522,Z 371.04,A -85,B 0,C 180,E1 -17284.862,E2 -17284.862} C_VEL
LIN {X 0,Y 283.905,Z 371.12,A -85,B 0,C 180,E1 -17286.046,E2 -17286.046} C_VEL
LIN {X 0,Y 281.057,Z 371.474,A -85,B 0,C 180,E1 -17287.973,E2 -17287.973} C_VEL
LIN {X 0,Y 278.597,Z 371.782,A -85,B 0,C 180,E1 -17289.539,E2 -17289.539} C_VEL
LIN {X 0,Y 277.525,Z 371.912,A -85,B 0,C 180,E1 -17290.753,E2 -17290.753} C_VEL
LIN {X 0,Y 277.432,Z 371.923,A -85,B 0,C 180,E1 -17291.164,E2 -17291.164} C_VEL
LIN {X 0,Y 277.435,Z 371.926,A -85,B 0,C 180,E1 -17295.723,E2 -17295.723} C_VEL
LIN {X 0,Y 277.337,Z 371.935,A -85,B 0,C 180,E1 -17300.351,E2 -17300.351} C_VEL
LIN {X 0,Y 277.31,Z 371.94,A -85,B 0,C 180,E1 -17304.171,E2 -17304.171} C_VEL
LIN {X 0,Y 277.315,Z 371.941,A -85,B 0,C 180,E1 -17307.505,E2 -17307.505} C_VEL
LIN {X 0,Y 277.264,Z 371.945,A -85,B 0,C 180,E1 -17310.483,E2 -17310.483} C_VEL
LIN {X 0,Y 277.247,Z 371.948,A -85,B 0,C 180,E1 -17313.896,E2 -17313.896} C_VEL
LIN {X 0,Y 277.286,Z 371.945,A -85,B 0,C 180,E1 -17317.467,E2 -17317.467} C_VEL
LIN {X 0,Y 277.289,Z 371.947,A -85,B 0,C 180,E1 -17321.223,E2 -17321.223} C_VEL
LIN {X 0,Y 277.283,Z 371.946,A -85,B 0,C 180,E1 -17325.21,E2 -17325.21} C_VEL
LIN {X 0,Y 277.291,Z 371.945,A -85,B 0,C 180,E1 -17329.496,E2 -17329.496} C_VEL
LIN {X 0,Y 277.287,Z 371.943,A -85,B 0,C 180,E1 -17332.536,E2 -17332.536} C_VEL
LIN {X 0,Y 277.354,Z 372.007,A -85,B 0,C 180,E1 -17336.163,E2 -17336.163} C_VEL
LIN {X 0,Y 280.417,Z 387.231,A -85,B 0,C 180,E1 -17340.597,E2 -17340.597} C_VEL
LIN {X 0,Y 281.397,Z 392.484,A -85,B 0,C 180,E1 -17342.079,E2 -17342.079} C_VEL
LIN {X 0,Y 280.464,Z 400.837,A -85,B 0,C 180,E1 -17344.318,E2 -17344.318} C_VEL
LIN {X 0,Y 279.895,Z 405.199,A -85,B 0,C 180,E1 -17345.477,E2 -17345.477} C_VEL
LIN {X 0,Y 281.291,Z 428.492,A -85,B 0,C 180,E1 -17346.493,E2 -17346.493} C_VEL
LIN {X 0,Y 283.743,Z 454.441,A -85,B 0,C 180,E1 -17347.62,E2 -17347.62} C_VEL
LIN {X 0,Y 281.654,Z 515.36,A -85,B 0,C 180,E1 -17350.031,E2 -17350.031} C_VEL
LIN {X 0,Y 280.83,Z 528.659,A -85,B 0,C 180,E1 -17350.826,E2 -17350.826} C_VEL
LIN {X 0,Y 279.883,Z 541.61,A -85,B 0,C 180,E1 -17351.898,E2 -17351.898} C_VEL
LIN {X 0,Y 279.054,Z 553.223,A -85,B 0,C 180,E1 -17353.144,E2 -17353.144} C_VEL
LIN {X 0,Y 278.139,Z 564.205,A -85,B 0,C 180,E1 -17354.616,E2 -17354.616} C_VEL
LIN {X 0,Y 277.31,Z 575.106,A -85,B 0,C 180,E1 -17356.444,E2 -17356.444} C_VEL
LIN {X 0,Y 276.707,Z 584.032,A -85,B 0,C 180,E1 -17358.278,E2 -17358.278} C_VEL
LIN {X 0,Y 276.246,Z 592.666,A -85,B 0,C 180,E1 -17360.483,E2 -17360.483} C_VEL
LIN {X 0,Y 276.101,Z 599.57,A -85,B 0,C 180,E1 -17362.69,E2 -17362.69} C_VEL
LIN {X 0,Y 276.089,Z 604.971,A -85,B 0,C 180,E1 -17364.89,E2 -17364.89} C_VEL
LIN {X 0,Y 276.139,Z 609.025,A -85,B 0,C 180,E1 -17367.084,E2 -17367.084} C_VEL
LIN {X 0,Y 276.251,Z 611.044,A -85,B 0,C 180,E1 -17368.544,E2 -17368.544} C_VEL
LIN {X 0,Y 276.229,Z 612.561,A -85,B 0,C 180,E1 -17370.002,E2 -17370.002} C_VEL
LIN {X 0,Y 275.919,Z 613.583,A -85,B 0,C 180,E1 -17371.461,E2 -17371.461} C_VEL
LIN {X 0,Y 275.717,Z 614.143,A -85,B 0,C 180,E1 -17372.924,E2 -17372.924} C_VEL
LIN {X 0,Y 275.567,Z 614.255,A -85,B 0,C 180,E1 -17374.39,E2 -17374.39} C_VEL
LIN {X 0,Y 275.532,Z 613.951,A -85,B 0,C 180,E1 -17375.858,E2 -17375.858} C_VEL
LIN {X 0,Y 275.511,Z 613.23,A -85,B 0,C 180,E1 -17377.329,E2 -17377.329} C_VEL
LIN {X 0,Y 275.693,Z 612.089,A -85,B 0,C 180,E1 -17378.8,E2 -17378.8} C_VEL
LIN {X 0,Y 276.004,Z 610.508,A -85,B 0,C 180,E1 -17380.269,E2 -17380.269} C_VEL
LIN {X 0,Y 276.819,Z 607.367,A -85,B 0,C 180,E1 -17382.464,E2 -17382.464} C_VEL
LIN {X 0,Y 278.2,Z 603.218,A -85,B 0,C 180,E1 -17384.634,E2 -17384.634} C_VEL
LIN {X 0,Y 280.122,Z 596.998,A -85,B 0,C 180,E1 -17387.147,E2 -17387.147} C_VEL
LIN {X 0,Y 282.945,Z 589.141,A -85,B 0,C 180,E1 -17389.594,E2 -17389.594} C_VEL
LIN {X 0,Y 285.896,Z 580.798,A -85,B 0,C 180,E1 -17391.639,E2 -17391.639} C_VEL
LIN {X 0,Y 289.321,Z 570.712,A -85,B 0,C 180,E1 -17393.63,E2 -17393.63} C_VEL
LIN {X 0,Y 292.612,Z 560.586,A -85,B 0,C 180,E1 -17395.236,E2 -17395.236} C_VEL
LIN {X 0,Y 296.214,Z 548.343,A -85,B 0,C 180,E1 -17396.796,E2 -17396.796} C_VEL
LIN {X 0,Y 299.605,Z 536.265,A -85,B 0,C 180,E1 -17397.981,E2 -17397.981} C_VEL
LIN {X 0,Y 302.992,Z 521.977,A -85,B 0,C 180,E1 -17399.057,E2 -17399.057} C_VEL
LIN {X 0,Y 305.694,Z 507.171,A -85,B 0,C 180,E1 -17399.909,E2 -17399.909} C_VEL
LIN {X 0,Y 311.7,Z 461.331,A -85,B 0,C 180,E1 -17401.886,E2 -17401.886} C_VEL
LIN {X 0,Y 311.79,Z 451.335,A -85,B 0,C 180,E1 -17402.679,E2 -17402.679} C_VEL
LIN {X 0,Y 311.265,Z 438.522,A -85,B 0,C 180,E1 -17403.993,E2 -17403.993} C_VEL
LIN {X 0,Y 310.862,Z 434.129,A -85,B 0,C 180,E1 -17404.551,E2 -17404.551} C_VEL
LIN {X 0,Y 308.516,Z 427.709,A -85,B 0,C 180,E1 -17406.152,E2 -17406.152} C_VEL
LIN {X 0,Y 306.543,Z 422.417,A -85,B 0,C 180,E1 -17407.759,E2 -17407.759} C_VEL
LIN {X 0,Y 303.758,Z 415.479,A -85,B 0,C 180,E1 -17410.772,E2 -17410.772} C_VEL
LIN {X 0,Y 302.268,Z 412.118,A -85,B 0,C 180,E1 -17413.583,E2 -17413.583} C_VEL
LIN {X 0,Y 302.089,Z 410.506,A -85,B 0,C 180,E1 -17415.921,E2 -17415.921} C_VEL
LIN {X 0,Y 302.71,Z 409.99,A -85,B 0,C 180,E1 -17417.984,E2 -17417.984} C_VEL
LIN {X 0,Y 303.457,Z 410.445,A -85,B 0,C 180,E1 -17419.383,E2 -17419.383} C_VEL
LIN {X 0,Y 306.03,Z 412.871,A -85,B 0,C 180,E1 -17422.236,E2 -17422.236} C_VEL
LIN {X 0,Y 308.708,Z 416.488,A -85,B 0,C 180,E1 -17424.327,E2 -17424.327} C_VEL
LIN {X 0,Y 311.421,Z 420.485,A -85,B 0,C 180,E1 -17426.014,E2 -17426.014} C_VEL
LIN {X 0,Y 314.167,Z 424.982,A -85,B 0,C 180,E1 -17427.488,E2 -17427.488} C_VEL
LIN {X 0,Y 315.421,Z 427.297,A -85,B 0,C 180,E1 -17428.108,E2 -17428.108} C_VEL
LIN {X 0,Y 308.14,Z 479.61,A -85,B 0,C 180,E1 -17430.37,E2 -17430.37} C_VEL
LIN {X 0,Y 306.173,Z 492.893,A -85,B 0,C 180,E1 -17431.181,E2 -17431.181} C_VEL
LIN {X 0,Y 303.721,Z 505.726,A -85,B 0,C 180,E1 -17432.222,E2 -17432.222} C_VEL
LIN {X 0,Y 300.606,Z 518.989,A -85,B 0,C 180,E1 -17433.627,E2 -17433.627} C_VEL
LIN {X 0,Y 297.431,Z 530.525,A -85,B 0,C 180,E1 -17435.202,E2 -17435.202} C_VEL
LIN {X 0,Y 294.364,Z 540.02,A -85,B 0,C 180,E1 -17436.8,E2 -17436.8} C_VEL
LIN {X 0,Y 291.565,Z 547.923,A -85,B 0,C 180,E1 -17438.433,E2 -17438.433} C_VEL
LIN {X 0,Y 288.563,Z 555.715,A -85,B 0,C 180,E1 -17440.434,E2 -17440.434} C_VEL
LIN {X 0,Y 285.506,Z 562.929,A -85,B 0,C 180,E1 -17442.819,E2 -17442.819} C_VEL
LIN {X 0,Y 283.261,Z 567.751,A -85,B 0,C 180,E1 -17444.899,E2 -17444.899} C_VEL
LIN {X 0,Y 281.302,Z 571.467,A -85,B 0,C 180,E1 -17447.005,E2 -17447.005} C_VEL
LIN {X 0,Y 280.143,Z 573.367,A -85,B 0,C 180,E1 -17448.422,E2 -17448.422} C_VEL
LIN {X 0,Y 279.077,Z 574.821,A -85,B 0,C 180,E1 -17449.847,E2 -17449.847} C_VEL
LIN {X 0,Y 278.275,Z 575.841,A -85,B 0,C 180,E1 -17451.284,E2 -17451.284} C_VEL
LIN {X 0,Y 277.621,Z 576.457,A -85,B 0,C 180,E1 -17452.728,E2 -17452.728} C_VEL
LIN {X 0,Y 277.197,Z 576.608,A -85,B 0,C 180,E1 -17454.179,E2 -17454.179} C_VEL
LIN {X 0,Y 276.801,Z 576.359,A -85,B 0,C 180,E1 -17455.631,E2 -17455.631} C_VEL
LIN {X 0,Y 276.358,Z 575.719,A -85,B 0,C 180,E1 -17457.084,E2 -17457.084} C_VEL
LIN {X 0,Y 275.999,Z 574.65,A -85,B 0,C 180,E1 -17458.541,E2 -17458.541} C_VEL
LIN {X 0,Y 275.815,Z 573.113,A -85,B 0,C 180,E1 -17460,E2 -17460} C_VEL
LIN {X 0,Y 275.725,Z 569.988,A -85,B 0,C 180,E1 -17462.191,E2 -17462.191} C_VEL
LIN {X 0,Y 275.935,Z 565.779,A -85,B 0,C 180,E1 -17464.382,E2 -17464.382} C_VEL
LIN {X 0,Y 276.113,Z 559.399,A -85,B 0,C 180,E1 -17466.927,E2 -17466.927} C_VEL
LIN {X 0,Y 276.545,Z 552.277,A -85,B 0,C 180,E1 -17469.139,E2 -17469.139} C_VEL
LIN {X 0,Y 277.181,Z 543.527,A -85,B 0,C 180,E1 -17471.332,E2 -17471.332} C_VEL
LIN {X 0,Y 277.946,Z 533.632,A -85,B 0,C 180,E1 -17473.34,E2 -17473.34} C_VEL
LIN {X 0,Y 278.883,Z 522.542,A -85,B 0,C 180,E1 -17475.156,E2 -17475.156} C_VEL
LIN {X 0,Y 279.759,Z 511.649,A -85,B 0,C 180,E1 -17476.604,E2 -17476.604} C_VEL
LIN {X 0,Y 280.453,Z 499.139,A -85,B 0,C 180,E1 -17477.933,E2 -17477.933} C_VEL
LIN {X 0,Y 281.189,Z 486.729,A -85,B 0,C 180,E1 -17478.961,E2 -17478.961} C_VEL
LIN {X 0,Y 281.876,Z 472.516,A -85,B 0,C 180,E1 -17479.812,E2 -17479.812} C_VEL
LIN {X 0,Y 283.804,Z 416.102,A -85,B 0,C 180,E1 -17482.017,E2 -17482.017} C_VEL
LIN {X 0,Y 284.525,Z 395.629,A -85,B 0,C 180,E1 -17482.798,E2 -17482.798} C_VEL
LIN {X 0,Y 277.341,Z 371.935,A -85,B 0,C 180,E1 -17484.081,E2 -17484.081} C_VEL
LIN {X 0,Y 277.332,Z 371.937,A -85,B 0,C 180,E1 -17487.505,E2 -17487.505} C_VEL
LIN {X 0,Y 277.278,Z 371.946,A -85,B 0,C 180,E1 -17490.481,E2 -17490.481} C_VEL
LIN {X 0,Y 277.252,Z 371.947,A -85,B 0,C 180,E1 -17493.895,E2 -17493.895} C_VEL
LIN {X 0,Y 277.277,Z 371.944,A -85,B 0,C 180,E1 -17497.468,E2 -17497.468} C_VEL
LIN {X 0,Y 277.214,Z 371.95,A -85,B 0,C 180,E1 -17501.236,E2 -17501.236} C_VEL
LIN {X 0,Y 277.206,Z 371.952,A -85,B 0,C 180,E1 -17505.225,E2 -17505.225} C_VEL
LIN {X 0,Y 277.227,Z 371.949,A -85,B 0,C 180,E1 -17509.511,E2 -17509.511} C_VEL
LIN {X 0,Y 277.278,Z 371.945,A -85,B 0,C 180,E1 -17512.531,E2 -17512.531} C_VEL
LIN {X 0,Y 277.251,Z 371.951,A -85,B 0,C 180,E1 -17516.103,E2 -17516.103} C_VEL
LIN {X 0,Y 277.265,Z 371.944,A -85,B 0,C 180,E1 -17519.537,E2 -17519.537} C_VEL
LIN {X 0,Y 277.361,Z 371.933,A -85,B 0,C 180,E1 -17522.863,E2 -17522.863} C_VEL
LIN {X 0,Y 277.333,Z 371.941,A -85,B 0,C 180,E1 -17526.078,E2 -17526.078} C_VEL
LIN {X 0,Y 277.348,Z 371.935,A -85,B 0,C 180,E1 -17530.765,E2 -17530.765} C_VEL
LIN {X 0,Y 277.438,Z 371.923,A -85,B 0,C 180,E1 -17535.324,E2 -17535.324} C_VEL
LIN {X 0,Y 277.464,Z 371.923,A -85,B 0,C 180,E1 -17539.785,E2 -17539.785} C_VEL
LIN {X 0,Y 277.643,Z 371.898,A -85,B 0,C 180,E1 -17542.727,E2 -17542.727} C_VEL
LIN {X 0,Y 277.824,Z 371.876,A -85,B 0,C 180,E1 -17548.549,E2 -17548.549} C_VEL
LIN {X 0,Y 277.823,Z 371.876,A -85,B 0,C 180,E1 -17551.448,E2 -17551.448} C_VEL
LIN {X 0,Y 277.654,Z 371.897,A -85,B 0,C 180,E1 -17557.269,E2 -17557.269} C_VEL
LIN {X 0,Y 277.506,Z 371.917,A -85,B 0,C 180,E1 -17560.21,E2 -17560.21} C_VEL
LIN {X 0,Y 277.433,Z 371.924,A -85,B 0,C 180,E1 -17564.672,E2 -17564.672} C_VEL
LIN {X 0,Y 277.343,Z 371.936,A -85,B 0,C 180,E1 -17569.232,E2 -17569.232} C_VEL
LIN {X 0,Y 277.317,Z 371.941,A -85,B 0,C 180,E1 -17574.169,E2 -17574.169} C_VEL
LIN {X 0,Y 277.323,Z 371.94,A -85,B 0,C 180,E1 -17577.504,E2 -17577.504} C_VEL
LIN {X 0,Y 277.268,Z 371.944,A -85,B 0,C 180,E1 -17580.48,E2 -17580.48} C_VEL
LIN {X 0,Y 277.25,Z 371.951,A -85,B 0,C 180,E1 -17583.893,E2 -17583.893} C_VEL
LIN {X 0,Y 277.286,Z 371.944,A -85,B 0,C 180,E1 -17587.464,E2 -17587.464} C_VEL
LIN {X 0,Y 277.261,Z 371.946,A -85,B 0,C 180,E1 -17591.225,E2 -17591.225} C_VEL
LIN {X 0,Y 277.282,Z 371.944,A -85,B 0,C 180,E1 -17595.207,E2 -17595.207} C_VEL
LIN {X 0,Y 277.289,Z 371.944,A -85,B 0,C 180,E1 -17599.493,E2 -17599.493} C_VEL
LIN {X 0,Y 277.283,Z 371.943,A -85,B 0,C 180,E1 -17602.533,E2 -17602.533} C_VEL
LIN {X 0,Y 277.247,Z 371.948,A -85,B 0,C 180,E1 -17606.104,E2 -17606.104} C_VEL
LIN {X 0,Y 277.253,Z 371.95,A -85,B 0,C 180,E1 -17609.538,E2 -17609.538} C_VEL
LIN {X 0,Y 277.354,Z 371.934,A -85,B 0,C 180,E1 -17612.864,E2 -17612.864} C_VEL
LIN {X 0,Y 277.321,Z 371.938,A -85,B 0,C 180,E1 -17616.079,E2 -17616.079} C_VEL
LIN {X 0,Y 277.336,Z 371.936,A -85,B 0,C 180,E1 -17620.766,E2 -17620.766} C_VEL
LIN {X 0,Y 277.426,Z 371.926,A -85,B 0,C 180,E1 -17625.326,E2 -17625.326} C_VEL
LIN {X 0,Y 277.498,Z 371.919,A -85,B 0,C 180,E1 -17629.789,E2 -17629.789} C_VEL
LIN {X 0,Y 277.644,Z 371.897,A -85,B 0,C 180,E1 -17632.729,E2 -17632.729} C_VEL
LIN {X 0,Y 277.816,Z 371.876,A -85,B 0,C 180,E1 -17638.551,E2 -17638.551} C_VEL
LIN {X 0,Y 277.814,Z 371.88,A -85,B 0,C 180,E1 -17641.45,E2 -17641.45} C_VEL
LIN {X 0,Y 277.645,Z 371.901,A -85,B 0,C 180,E1 -17647.271,E2 -17647.271} C_VEL
LIN {X 0,Y 277.498,Z 371.915,A -85,B 0,C 180,E1 -17650.212,E2 -17650.212} C_VEL
LIN {X 0,Y 277.432,Z 371.923,A -85,B 0,C 180,E1 -17651.164,E2 -17651.164} C_VEL
LIN {X 0,Y 276.741,Z 372.012,A -85,B 0,C 180,E1 -17652.377,E2 -17652.377} C_VEL
LIN {X 0,Y 273.863,Z 372.37,A -85,B 0,C 180,E1 -17654.351,E2 -17654.351} C_VEL
LIN {X 0,Y 271.425,Z 372.673,A -85,B 0,C 180,E1 -17655.956,E2 -17655.956} C_VEL
LIN {X 0,Y 270.372,Z 372.807,A -85,B 0,C 180,E1 -17657.2,E2 -17657.2} C_VEL
LIN {X 0,Y 270.281,Z 372.812,A -85,B 0,C 180,E1 -17657.621,E2 -17657.621} C_VEL
LIN {X 0,Y 270.214,Z 372.827,A -85,B 0,C 180,E1 -17661.354,E2 -17661.354} C_VEL
LIN {X 0,Y 270.266,Z 372.817,A -85,B 0,C 180,E1 -17664.587,E2 -17664.587} C_VEL
LIN {X 0,Y 270.262,Z 372.816,A -85,B 0,C 180,E1 -17667.91,E2 -17667.91} C_VEL
LIN {X 0,Y 270.176,Z 372.833,A -85,B 0,C 180,E1 -17671.349,E2 -17671.349} C_VEL
LIN {X 0,Y 270.209,Z 372.826,A -85,B 0,C 180,E1 -17674.905,E2 -17674.905} C_VEL
LIN {X 0,Y 270.246,Z 372.819,A -85,B 0,C 180,E1 -17678.727,E2 -17678.727} C_VEL
LIN {X 0,Y 270.251,Z 372.819,A -85,B 0,C 180,E1 -17682.543,E2 -17682.543} C_VEL
LIN {X 0,Y 270.228,Z 372.821,A -85,B 0,C 180,E1 -17686.737,E2 -17686.737} C_VEL
LIN {X 0,Y 270.245,Z 372.823,A -85,B 0,C 180,E1 -17689.45,E2 -17689.45} C_VEL
LIN {X 0,Y 270.254,Z 372.818,A -85,B 0,C 180,E1 -17693.723,E2 -17693.723} C_VEL
LIN {X 0,Y 270.339,Z 372.955,A -85,B 0,C 180,E1 -17696.006,E2 -17696.006} C_VEL
LIN {X 0,Y 273.575,Z 389.217,A -85,B 0,C 180,E1 -17700.862,E2 -17700.862} C_VEL
LIN {X 0,Y 274.337,Z 393.631,A -85,B 0,C 180,E1 -17702.128,E2 -17702.128} C_VEL
LIN {X 0,Y 272.915,Z 404.699,A -85,B 0,C 180,E1 -17705.163,E2 -17705.163} C_VEL
LIN {X 0,Y 274.132,Z 426.881,A -85,B 0,C 180,E1 -17706.164,E2 -17706.164} C_VEL
LIN {X 0,Y 276.731,Z 454.494,A -85,B 0,C 180,E1 -17707.405,E2 -17707.405} C_VEL
LIN {X 0,Y 274.606,Z 514.847,A -85,B 0,C 180,E1 -17709.887,E2 -17709.887} C_VEL
LIN {X 0,Y 273.782,Z 528.044,A -85,B 0,C 180,E1 -17710.703,E2 -17710.703} C_VEL
LIN {X 0,Y 273.004,Z 539.084,A -85,B 0,C 180,E1 -17711.62,E2 -17711.62} C_VEL
LIN {X 0,Y 272.09,Z 551.508,A -85,B 0,C 180,E1 -17712.953,E2 -17712.953} C_VEL
LIN {X 0,Y 271.085,Z 563.554,A -85,B 0,C 180,E1 -17714.591,E2 -17714.591} C_VEL
LIN {X 0,Y 270.239,Z 574.469,A -85,B 0,C 180,E1 -17716.466,E2 -17716.466} C_VEL
LIN {X 0,Y 269.645,Z 583.387,A -85,B 0,C 180,E1 -17718.348,E2 -17718.348} C_VEL
LIN {X 0,Y 269.206,Z 592.023,A -85,B 0,C 180,E1 -17720.611,E2 -17720.611} C_VEL
LIN {X 0,Y 269.079,Z 599.227,A -85,B 0,C 180,E1 -17722.987,E2 -17722.987} C_VEL
LIN {X 0,Y 269.078,Z 605.069,A -85,B 0,C 180,E1 -17725.508,E2 -17725.508} C_VEL
LIN {X 0,Y 269.135,Z 608.899,A -85,B 0,C 180,E1 -17727.757,E2 -17727.757} C_VEL
LIN {X 0,Y 269.196,Z 611.554,A -85,B 0,C 180,E1 -17730.002,E2 -17730.002} C_VEL
LIN {X 0,Y 268.894,Z 612.665,A -85,B 0,C 180,E1 -17731.499,E2 -17731.499} C_VEL
LIN {X 0,Y 268.656,Z 613.343,A -85,B 0,C 180,E1 -17733.001,E2 -17733.001} C_VEL
LIN {X 0,Y 268.451,Z 613.447,A -85,B 0,C 180,E1 -17735.823,E2 -17735.823} C_VEL
LIN {X 0,Y 268.458,Z 612.762,A -85,B 0,C 180,E1 -17737.523,E2 -17737.523} C_VEL
LIN {X 0,Y 268.97,Z 610.319,A -85,B 0,C 180,E1 -17740.541,E2 -17740.541} C_VEL
LIN {X 0,Y 269.877,Z 607.367,A -85,B 0,C 180,E1 -17742.79,E2 -17742.79} C_VEL
LIN {X 0,Y 271.323,Z 603.441,A -85,B 0,C 180,E1 -17745.014,E2 -17745.014} C_VEL
LIN {X 0,Y 273.078,Z 598.477,A -85,B 0,C 180,E1 -17747.217,E2 -17747.217} C_VEL
LIN {X 0,Y 275.443,Z 592.36,A -85,B 0,C 180,E1 -17749.374,E2 -17749.374} C_VEL
LIN {X 0,Y 278.349,Z 584.935,A -85,B 0,C 180,E1 -17751.477,E2 -17751.477} C_VEL
LIN {X 0,Y 281.731,Z 575.94,A -85,B 0,C 180,E1 -17753.526,E2 -17753.526} C_VEL
LIN {X 0,Y 285.645,Z 565.057,A -85,B 0,C 180,E1 -17755.505,E2 -17755.505} C_VEL
LIN {X 0,Y 289.728,Z 552.808,A -85,B 0,C 180,E1 -17757.25,E2 -17757.25} C_VEL
LIN {X 0,Y 293.561,Z 540.489,A -85,B 0,C 180,E1 -17758.609,E2 -17758.609} C_VEL
LIN {X 0,Y 297.256,Z 526.753,A -85,B 0,C 180,E1 -17759.77,E2 -17759.77} C_VEL
LIN {X 0,Y 300.423,Z 512.535,A -85,B 0,C 180,E1 -17760.684,E2 -17760.684} C_VEL
LIN {X 0,Y 302.975,Z 496.604,A -85,B 0,C 180,E1 -17761.463,E2 -17761.463} C_VEL
LIN {X 0,Y 307.688,Z 462.812,A -85,B 0,C 180,E1 -17762.931,E2 -17762.931} C_VEL
LIN {X 0,Y 307.912,Z 453.072,A -85,B 0,C 180,E1 -17763.744,E2 -17763.744} C_VEL
LIN {X 0,Y 307.629,Z 440.879,A -85,B 0,C 180,E1 -17765.058,E2 -17765.058} C_VEL
LIN {X 0,Y 307.4,Z 438.582,A -85,B 0,C 180,E1 -17765.389,E2 -17765.389} C_VEL
LIN {X 0,Y 305.586,Z 433.196,A -85,B 0,C 180,E1 -17766.797,E2 -17766.797} C_VEL
LIN {X 0,Y 303.913,Z 428.336,A -85,B 0,C 180,E1 -17768.324,E2 -17768.324} C_VEL
LIN {X 0,Y 301.673,Z 422.059,A -85,B 0,C 180,E1 -17771.084,E2 -17771.084} C_VEL
LIN {X 0,Y 300.38,Z 418.763,A -85,B 0,C 180,E1 -17773.914,E2 -17773.914} C_VEL
LIN {X 0,Y 300.388,Z 417.153,A -85,B 0,C 180,E1 -17776.495,E2 -17776.495} C_VEL
LIN {X 0,Y 301.369,Z 416.985,A -85,B 0,C 180,E1 -17778.851,E2 -17778.851} C_VEL
LIN {X 0,Y 303.896,Z 419.503,A -85,B 0,C 180,E1 -17781.977,E2 -17781.977} C_VEL
LIN {X 0,Y 306.413,Z 423.134,A -85,B 0,C 180,E1 -17784.078,E2 -17784.078} C_VEL
LIN {X 0,Y 308.95,Z 427.034,A -85,B 0,C 180,E1 -17785.746,E2 -17785.746} C_VEL
LIN {X 0,Y 311.37,Z 431.301,A -85,B 0,C 180,E1 -17787.124,E2 -17787.124} C_VEL
LIN {X 0,Y 303.888,Z 481.574,A -85,B 0,C 180,E1 -17789.356,E2 -17789.356} C_VEL
LIN {X 0,Y 301.746,Z 494.492,A -85,B 0,C 180,E1 -17790.176,E2 -17790.176} C_VEL
LIN {X 0,Y 299.186,Z 506.933,A -85,B 0,C 180,E1 -17791.213,E2 -17791.213} C_VEL
LIN {X 0,Y 295.544,Z 521.109,A -85,B 0,C 180,E1 -17792.757,E2 -17792.757} C_VEL
LIN {X 0,Y 291.855,Z 533.275,A -85,B 0,C 180,E1 -17794.504,E2 -17794.504} C_VEL
LIN {X 0,Y 288.297,Z 543.189,A -85,B 0,C 180,E1 -17796.282,E2 -17796.282} C_VEL
LIN {X 0,Y 284.807,Z 551.983,A -85,B 0,C 180,E1 -17798.275,E2 -17798.275} C_VEL
LIN {X 0,Y 281.715,Z 559.126,A -85,B 0,C 180,E1 -17800.319,E2 -17800.319} C_VEL
LIN {X 0,Y 278.983,Z 564.852,A -85,B 0,C 180,E1 -17802.404,E2 -17802.404} C_VEL
LIN {X 0,Y 276.595,Z 569.384,A -85,B 0,C 180,E1 -17804.526,E2 -17804.526} C_VEL
LIN {X 0,Y 274.544,Z 572.841,A -85,B 0,C 180,E1 -17806.68,E2 -17806.68} C_VEL
LIN {X 0,Y 273.303,Z 574.586,A -85,B 0,C 180,E1 -17808.128,E2 -17808.128} C_VEL
LIN {X 0,Y 272.193,Z 575.918,A -85,B 0,C 180,E1 -17809.587,E2 -17809.587} C_VEL
LIN {X 0,Y 271.341,Z 576.795,A -85,B 0,C 180,E1 -17811.059,E2 -17811.059} C_VEL
LIN {X 0,Y 270.626,Z 577.239,A -85,B 0,C 180,E1 -17812.539,E2 -17812.539} C_VEL
LIN {X 0,Y 270.18,Z 577.27,A -85,B 0,C 180,E1 -17814.027,E2 -17814.027} C_VEL
LIN {X 0,Y 269.764,Z 576.914,A -85,B 0,C 180,E1 -17815.517,E2 -17815.517} C_VEL
LIN {X 0,Y 269.293,Z 576.126,A -85,B 0,C 180,E1 -17817.008,E2 -17817.008} C_VEL
LIN {X 0,Y 268.906,Z 574.902,A -85,B 0,C 180,E1 -17818.502,E2 -17818.502} C_VEL
LIN {X 0,Y 268.649,Z 572.26,A -85,B 0,C 180,E1 -17820.749,E2 -17820.749} C_VEL
LIN {X 0,Y 268.698,Z 568.577,A -85,B 0,C 180,E1 -17822.998,E2 -17822.998} C_VEL
LIN {X 0,Y 268.888,Z 563.758,A -85,B 0,C 180,E1 -17825.249,E2 -17825.249} C_VEL
LIN {X 0,Y 269.216,Z 556.508,A -85,B 0,C 180,E1 -17827.877,E2 -17827.877} C_VEL
LIN {X 0,Y 269.717,Z 548.609,A -85,B 0,C 180,E1 -17830.13,E2 -17830.13} C_VEL
LIN {X 0,Y 270.452,Z 538.859,A -85,B 0,C 180,E1 -17832.379,E2 -17832.379} C_VEL
LIN {X 0,Y 271.404,Z 527.691,A -85,B 0,C 180,E1 -17834.432,E2 -17834.432} C_VEL
LIN {X 0,Y 272.241,Z 516.369,A -85,B 0,C 180,E1 -17836.112,E2 -17836.112} C_VEL
LIN {X 0,Y 272.963,Z 506.026,A -85,B 0,C 180,E1 -17837.362,E2 -17837.362} C_VEL
LIN {X 0,Y 273.785,Z 493.028,A -85,B 0,C 180,E1 -17838.619,E2 -17838.619} C_VEL
LIN {X 0,Y 274.573,Z 478.881,A -85,B 0,C 180,E1 -17839.63,E2 -17839.63} C_VEL
LIN {X 0,Y 275.035,Z 464.795,A -85,B 0,C 180,E1 -17840.326,E2 -17840.326} C_VEL
LIN {X 0,Y 277.482,Z 396.674,A -85,B 0,C 180,E1 -17843.034,E2 -17843.034} C_VEL
LIN {X 0,Y 270.291,Z 372.815,A -85,B 0,C 180,E1 -17844.343,E2 -17844.343} C_VEL
LIN {X 0,Y 270.278,Z 372.817,A -85,B 0,C 180,E1 -17847.908,E2 -17847.908} C_VEL
LIN {X 0,Y 270.19,Z 372.826,A -85,B 0,C 180,E1 -17851.347,E2 -17851.347} C_VEL
LIN {X 0,Y 270.208,Z 372.825,A -85,B 0,C 180,E1 -17854.905,E2 -17854.905} C_VEL
LIN {X 0,Y 270.203,Z 372.826,A -85,B 0,C 180,E1 -17858.709,E2 -17858.709} C_VEL
LIN {X 0,Y 270.177,Z 372.83,A -85,B 0,C 180,E1 -17862.557,E2 -17862.557} C_VEL
LIN {X 0,Y 270.17,Z 372.83,A -85,B 0,C 180,E1 -17866.75,E2 -17866.75} C_VEL
LIN {X 0,Y 270.178,Z 372.827,A -85,B 0,C 180,E1 -17869.433,E2 -17869.433} C_VEL
LIN {X 0,Y 270.248,Z 372.82,A -85,B 0,C 180,E1 -17873.724,E2 -17873.724} C_VEL
LIN {X 0,Y 270.207,Z 372.824,A -85,B 0,C 180,E1 -17876.891,E2 -17876.891} C_VEL
LIN {X 0,Y 270.223,Z 372.825,A -85,B 0,C 180,E1 -17880.384,E2 -17880.384} C_VEL
LIN {X 0,Y 270.266,Z 372.819,A -85,B 0,C 180,E1 -17883.762,E2 -17883.762} C_VEL
LIN {X 0,Y 270.236,Z 372.819,A -85,B 0,C 180,E1 -17887.037,E2 -17887.037} C_VEL
LIN {X 0,Y 270.305,Z 372.816,A -85,B 0,C 180,E1 -17890.243,E2 -17890.243} C_VEL
LIN {X 0,Y 270.406,Z 372.799,A -85,B 0,C 180,E1 -17894.934,E2 -17894.934} C_VEL
LIN {X 0,Y 270.415,Z 372.799,A -85,B 0,C 180,E1 -17899.516,E2 -17899.516} C_VEL
LIN {X 0,Y 270.601,Z 372.776,A -85,B 0,C 180,E1 -17902.537,E2 -17902.537} C_VEL
LIN {X 0,Y 270.789,Z 372.753,A -85,B 0,C 180,E1 -17908.511,E2 -17908.511} C_VEL
LIN {X 0,Y 270.789,Z 372.753,A -85,B 0,C 180,E1 -17911.485,E2 -17911.485} C_VEL
LIN {X 0,Y 270.612,Z 372.775,A -85,B 0,C 180,E1 -17917.459,E2 -17917.459} C_VEL
LIN {X 0,Y 270.441,Z 372.796,A -85,B 0,C 180,E1 -17920.479,E2 -17920.479} C_VEL
LIN {X 0,Y 270.402,Z 372.799,A -85,B 0,C 180,E1 -17925.063,E2 -17925.063} C_VEL
LIN {X 0,Y 270.299,Z 372.816,A -85,B 0,C 180,E1 -17929.754,E2 -17929.754} C_VEL
LIN {X 0,Y 270.271,Z 372.816,A -85,B 0,C 180,E1 -17934.584,E2 -17934.584} C_VEL
LIN {X 0,Y 270.267,Z 372.821,A -85,B 0,C 180,E1 -17937.907,E2 -17937.907} C_VEL
LIN {X 0,Y 270.181,Z 372.827,A -85,B 0,C 180,E1 -17941.346,E2 -17941.346} C_VEL
LIN {X 0,Y 270.211,Z 372.824,A -85,B 0,C 180,E1 -17944.902,E2 -17944.902} C_VEL
LIN {X 0,Y 270.217,Z 372.822,A -85,B 0,C 180,E1 -17948.715,E2 -17948.715} C_VEL
LIN {X 0,Y 270.225,Z 372.822,A -85,B 0,C 180,E1 -17952.545,E2 -17952.545} C_VEL
LIN {X 0,Y 270.229,Z 372.821,A -85,B 0,C 180,E1 -17956.734,E2 -17956.734} C_VEL
LIN {X 0,Y 270.243,Z 372.821,A -85,B 0,C 180,E1 -17959.447,E2 -17959.447} C_VEL
LIN {X 0,Y 270.25,Z 372.823,A -85,B 0,C 180,E1 -17963.72,E2 -17963.72} C_VEL
LIN {X 0,Y 270.196,Z 372.824,A -85,B 0,C 180,E1 -17966.892,E2 -17966.892} C_VEL
LIN {X 0,Y 270.228,Z 372.822,A -85,B 0,C 180,E1 -17970.387,E2 -17970.387} C_VEL
LIN {X 0,Y 270.258,Z 372.821,A -85,B 0,C 180,E1 -17973.763,E2 -17973.763} C_VEL
LIN {X 0,Y 270.224,Z 372.822,A -85,B 0,C 180,E1 -17977.038,E2 -17977.038} C_VEL
LIN {X 0,Y 270.293,Z 372.814,A -85,B 0,C 180,E1 -17980.244,E2 -17980.244} C_VEL
LIN {X 0,Y 270.394,Z 372.8,A -85,B 0,C 180,E1 -17984.935,E2 -17984.935} C_VEL
LIN {X 0,Y 270.433,Z 372.801,A -85,B 0,C 180,E1 -17989.519,E2 -17989.519} C_VEL
LIN {X 0,Y 270.602,Z 372.774,A -85,B 0,C 180,E1 -17992.539,E2 -17992.539} C_VEL
LIN {X 0,Y 270.782,Z 372.753,A -85,B 0,C 180,E1 -17998.513,E2 -17998.513} C_VEL
LIN {X 0,Y 270.78,Z 372.756,A -85,B 0,C 180,E1 -18001.487,E2 -18001.487} C_VEL
LIN {X 0,Y 270.603,Z 372.779,A -85,B 0,C 180,E1 -18007.462,E2 -18007.462} C_VEL
LIN {X 0,Y 270.433,Z 372.794,A -85,B 0,C 180,E1 -18010.482,E2 -18010.482} C_VEL
LIN {X 0,Y 270.394,Z 372.803,A -85,B 0,C 180,E1 -18015.065,E2 -18015.065} C_VEL
LIN {X 0,Y 270.281,Z 372.812,A -85,B 0,C 180,E1 -18017.621,E2 -18017.621} C_VEL
LIN {X 0,Y 269.588,Z 372.903,A -85,B 0,C 180,E1 -18018.865,E2 -18018.865} C_VEL
LIN {X 0,Y 266.692,Z 373.264,A -85,B 0,C 180,E1 -18020.891,E2 -18020.891} C_VEL
LIN {X 0,Y 264.263,Z 373.567,A -85,B 0,C 180,E1 -18022.538,E2 -18022.538} C_VEL
LIN {X 0,Y 263.251,Z 373.693,A -85,B 0,C 180,E1 -18023.816,E2 -18023.816} C_VEL
LIN {X 0,Y 263.184,Z 373.699,A -85,B 0,C 180,E1 -18024.248,E2 -18024.248} C_VEL
LIN {X 0,Y 263.188,Z 373.697,A -85,B 0,C 180,E1 -18028.216,E2 -18028.216} C_VEL
LIN {X 0,Y 263.126,Z 373.706,A -85,B 0,C 180,E1 -18032.289,E2 -18032.289} C_VEL
LIN {X 0,Y 263.184,Z 373.698,A -85,B 0,C 180,E1 -18035.979,E2 -18035.979} C_VEL
LIN {X 0,Y 263.187,Z 373.699,A -85,B 0,C 180,E1 -18039.858,E2 -18039.858} C_VEL
LIN {X 0,Y 263.186,Z 373.699,A -85,B 0,C 180,E1 -18043.971,E2 -18043.971} C_VEL
LIN {X 0,Y 263.208,Z 373.696,A -85,B 0,C 180,E1 -18048.387,E2 -18048.387} C_VEL
LIN {X 0,Y 263.203,Z 373.7,A -85,B 0,C 180,E1 -18053.231,E2 -18053.231} C_VEL
LIN {X 0,Y 263.283,Z 373.839,A -85,B 0,C 180,E1 -18055.844,E2 -18055.844} C_VEL
LIN {X 0,Y 266.358,Z 389.196,A -85,B 0,C 180,E1 -18060.543,E2 -18060.543} C_VEL
LIN {X 0,Y 267.253,Z 394.728,A -85,B 0,C 180,E1 -18062.177,E2 -18062.177} C_VEL
LIN {X 0,Y 265.923,Z 404.529,A -85,B 0,C 180,E1 -18064.893,E2 -18064.893} C_VEL
LIN {X 0,Y 267.142,Z 427.309,A -85,B 0,C 180,E1 -18065.931,E2 -18065.931} C_VEL
LIN {X 0,Y 269.716,Z 454.561,A -85,B 0,C 180,E1 -18067.197,E2 -18067.197} C_VEL
LIN {X 0,Y 267.539,Z 514.978,A -85,B 0,C 180,E1 -18069.783,E2 -18069.783} C_VEL
LIN {X 0,Y 266.672,Z 528.545,A -85,B 0,C 180,E1 -18070.668,E2 -18070.668} C_VEL
LIN {X 0,Y 265.791,Z 540.237,A -85,B 0,C 180,E1 -18071.707,E2 -18071.707} C_VEL
LIN {X 0,Y 264.784,Z 553.448,A -85,B 0,C 180,E1 -18073.225,E2 -18073.225} C_VEL
LIN {X 0,Y 263.81,Z 565.124,A -85,B 0,C 180,E1 -18074.947,E2 -18074.947} C_VEL
LIN {X 0,Y 263.049,Z 575.679,A -85,B 0,C 180,E1 -18076.876,E2 -18076.876} C_VEL
LIN {X 0,Y 262.422,Z 585.772,A -85,B 0,C 180,E1 -18079.197,E2 -18079.197} C_VEL
LIN {X 0,Y 262.128,Z 593.825,A -85,B 0,C 180,E1 -18081.522,E2 -18081.522} C_VEL
LIN {X 0,Y 262.079,Z 600.173,A -85,B 0,C 180,E1 -18083.844,E2 -18083.844} C_VEL
LIN {X 0,Y 262.108,Z 605.092,A -85,B 0,C 180,E1 -18086.158,E2 -18086.158} C_VEL
LIN {X 0,Y 262.184,Z 608.726,A -85,B 0,C 180,E1 -18088.466,E2 -18088.466} C_VEL
LIN {X 0,Y 262.169,Z 610.499,A -85,B 0,C 180,E1 -18090.002,E2 -18090.002} C_VEL
LIN {X 0,Y 261.867,Z 611.727,A -85,B 0,C 180,E1 -18091.54,E2 -18091.54} C_VEL
LIN {X 0,Y 261.618,Z 612.497,A -85,B 0,C 180,E1 -18093.082,E2 -18093.082} C_VEL
LIN {X 0,Y 261.382,Z 612.825,A -85,B 0,C 180,E1 -18095.813,E2 -18095.813} C_VEL
LIN {X 0,Y 261.381,Z 612.297,A -85,B 0,C 180,E1 -18097.728,E2 -18097.728} C_VEL
LIN {X 0,Y 261.954,Z 610.069,A -85,B 0,C 180,E1 -18100.826,E2 -18100.826} C_VEL
LIN {X 0,Y 262.92,Z 607.346,A -85,B 0,C 180,E1 -18103.135,E2 -18103.135} C_VEL
LIN {X 0,Y 264.465,Z 603.672,A -85,B 0,C 180,E1 -18105.413,E2 -18105.413} C_VEL
LIN {X 0,Y 266.979,Z 597.185,A -85,B 0,C 180,E1 -18108.416,E2 -18108.416} C_VEL
LIN {X 0,Y 270.188,Z 589.821,A -85,B 0,C 180,E1 -18110.958,E2 -18110.958} C_VEL
LIN {X 0,Y 274.169,Z 580.621,A -85,B 0,C 180,E1 -18113.413,E2 -18113.413} C_VEL
LIN {X 0,Y 278.046,Z 570.966,A -85,B 0,C 180,E1 -18115.45,E2 -18115.45} C_VEL
LIN {X 0,Y 282.529,Z 559.214,A -85,B 0,C 180,E1 -18117.401,E2 -18117.401} C_VEL
LIN {X 0,Y 286.2,Z 548.53,A -85,B 0,C 180,E1 -18118.812,E2 -18118.812} C_VEL
LIN {X 0,Y 290.439,Z 535.44,A -85,B 0,C 180,E1 -18120.141,E2 -18120.141} C_VEL
LIN {X 0,Y 294.159,Z 521.796,A -85,B 0,C 180,E1 -18121.21,E2 -18121.21} C_VEL
LIN {X 0,Y 297.385,Z 506.683,A -85,B 0,C 180,E1 -18122.124,E2 -18122.124} C_VEL
LIN {X 0,Y 303.9,Z 464.354,A -85,B 0,C 180,E1 -18124.023,E2 -18124.023} C_VEL
LIN {X 0,Y 304.27,Z 455.302,A -85,B 0,C 180,E1 -18124.809,E2 -18124.809} C_VEL
LIN {X 0,Y 304.221,Z 443.648,A -85,B 0,C 180,E1 -18126.123,E2 -18126.123} C_VEL
LIN {X 0,Y 302.763,Z 438.804,A -85,B 0,C 180,E1 -18127.43,E2 -18127.43} C_VEL
LIN {X 0,Y 301.391,Z 434.35,A -85,B 0,C 180,E1 -18128.866,E2 -18128.866} C_VEL
LIN {X 0,Y 299.554,Z 428.518,A -85,B 0,C 180,E1 -18131.489,E2 -18131.489} C_VEL
LIN {X 0,Y 298.532,Z 425.556,A -85,B 0,C 180,E1 -18134.089,E2 -18134.089} C_VEL
LIN {X 0,Y 298.618,Z 423.987,A -85,B 0,C 180,E1 -18136.613,E2 -18136.613} C_VEL
LIN {X 0,Y 299.615,Z 423.905,A -85,B 0,C 180,E1 -18138.944,E2 -18138.944} C_VEL
LIN {X 0,Y 301.867,Z 426.293,A -85,B 0,C 180,E1 -18141.81,E2 -18141.81} C_VEL
LIN {X 0,Y 304.02,Z 429.554,A -85,B 0,C 180,E1 -18143.727,E2 -18143.727} C_VEL
LIN {X 0,Y 306.439,Z 433.453,A -85,B 0,C 180,E1 -18145.421,E2 -18145.421} C_VEL
LIN {X 0,Y 307.552,Z 435.545,A -85,B 0,C 180,E1 -18146.131,E2 -18146.131} C_VEL
LIN {X 0,Y 300.237,Z 481.098,A -85,B 0,C 180,E1 -18148.169,E2 -18148.169} C_VEL
LIN {X 0,Y 297.87,Z 494.762,A -85,B 0,C 180,E1 -18149.026,E2 -18149.026} C_VEL
LIN {X 0,Y 295.22,Z 506.623,A -85,B 0,C 180,E1 -18150.005,E2 -18150.005} C_VEL
LIN {X 0,Y 292.138,Z 518.284,A -85,B 0,C 180,E1 -18151.24,E2 -18151.24} C_VEL
LIN {X 0,Y 288.813,Z 528.997,A -85,B 0,C 180,E1 -18152.657,E2 -18152.657} C_VEL
LIN {X 0,Y 284.934,Z 539.781,A -85,B 0,C 180,E1 -18154.428,E2 -18154.428} C_VEL
LIN {X 0,Y 281.004,Z 549.322,A -85,B 0,C 180,E1 -18156.411,E2 -18156.411} C_VEL
LIN {X 0,Y 277.484,Z 557.065,A -85,B 0,C 180,E1 -18158.454,E2 -18158.454} C_VEL
LIN {X 0,Y 274.356,Z 563.302,A -85,B 0,C 180,E1 -18160.548,E2 -18160.548} C_VEL
LIN {X 0,Y 271.567,Z 568.312,A -85,B 0,C 180,E1 -18162.685,E2 -18162.685} C_VEL
LIN {X 0,Y 269.161,Z 572.205,A -85,B 0,C 180,E1 -18164.864,E2 -18164.864} C_VEL
LIN {X 0,Y 267.797,Z 574.211,A -85,B 0,C 180,E1 -18166.338,E2 -18166.338} C_VEL
LIN {X 0,Y 266.47,Z 575.828,A -85,B 0,C 180,E1 -18167.819,E2 -18167.819} C_VEL
LIN {X 0,Y 265.315,Z 576.969,A -85,B 0,C 180,E1 -18169.314,E2 -18169.314} C_VEL
LIN {X 0,Y 263.637,Z 578.017,A -85,B 0,C 180,E1 -18172.34,E2 -18172.34} C_VEL
LIN {X 0,Y 263.167,Z 577.923,A -85,B 0,C 180,E1 -18173.868,E2 -18173.868} C_VEL
LIN {X 0,Y 262.71,Z 577.394,A -85,B 0,C 180,E1 -18175.397,E2 -18175.397} C_VEL
LIN {X 0,Y 262.212,Z 576.467,A -85,B 0,C 180,E1 -18176.927,E2 -18176.927} C_VEL
LIN {X 0,Y 261.813,Z 575.134,A -85,B 0,C 180,E1 -18178.462,E2 -18178.462} C_VEL
LIN {X 0,Y 261.556,Z 572.279,A -85,B 0,C 180,E1 -18180.77,E2 -18180.77} C_VEL
LIN {X 0,Y 261.624,Z 568.386,A -85,B 0,C 180,E1 -18183.08,E2 -18183.08} C_VEL
LIN {X 0,Y 261.787,Z 563.332,A -85,B 0,C 180,E1 -18185.391,E2 -18185.391} C_VEL
LIN {X 0,Y 262.177,Z 555.734,A -85,B 0,C 180,E1 -18188.09,E2 -18188.09} C_VEL
LIN {X 0,Y 262.694,Z 547.56,A -85,B 0,C 180,E1 -18190.404,E2 -18190.404} C_VEL
LIN {X 0,Y 263.483,Z 537.337,A -85,B 0,C 180,E1 -18192.712,E2 -18192.712} C_VEL
LIN {X 0,Y 264.371,Z 526.897,A -85,B 0,C 180,E1 -18194.628,E2 -18194.628} C_VEL
LIN {X 0,Y 265.28,Z 515.259,A -85,B 0,C 180,E1 -18196.349,E2 -18196.349} C_VEL
LIN {X 0,Y 266.047,Z 503.734,A -85,B 0,C 180,E1 -18197.73,E2 -18197.73} C_VEL
LIN {X 0,Y 266.923,Z 489.793,A -85,B 0,C 180,E1 -18199.016,E2 -18199.016} C_VEL
LIN {X 0,Y 267.579,Z 476.684,A -85,B 0,C 180,E1 -18199.915,E2 -18199.915} C_VEL
LIN {X 0,Y 268.343,Z 455.937,A -85,B 0,C 180,E1 -18200.856,E2 -18200.856} C_VEL
LIN {X 0,Y 270.506,Z 397.995,A -85,B 0,C 180,E1 -18203.254,E2 -18203.254} C_VEL
LIN {X 0,Y 263.238,Z 373.694,A -85,B 0,C 180,E1 -18204.612,E2 -18204.612} C_VEL
LIN {X 0,Y 263.186,Z 373.701,A -85,B 0,C 180,E1 -18208.729,E2 -18208.729} C_VEL
LIN {X 0,Y 263.139,Z 373.707,A -85,B 0,C 180,E1 -18212.287,E2 -18212.287} C_VEL
LIN {X 0,Y 263.169,Z 373.703,A -85,B 0,C 180,E1 -18215.981,E2 -18215.981} C_VEL
LIN {X 0,Y 263.111,Z 373.71,A -85,B 0,C 180,E1 -18219.871,E2 -18219.871} C_VEL
LIN {X 0,Y 263.127,Z 373.708,A -85,B 0,C 180,E1 -18223.983,E2 -18223.983} C_VEL
LIN {X 0,Y 263.129,Z 373.708,A -85,B 0,C 180,E1 -18228.405,E2 -18228.405} C_VEL
LIN {X 0,Y 263.198,Z 373.697,A -85,B 0,C 180,E1 -18233.232,E2 -18233.232} C_VEL
LIN {X 0,Y 263.172,Z 373.703,A -85,B 0,C 180,E1 -18235.887,E2 -18235.887} C_VEL
LIN {X 0,Y 263.152,Z 373.701,A -85,B 0,C 180,E1 -18239.505,E2 -18239.505} C_VEL
LIN {X 0,Y 263.195,Z 373.698,A -85,B 0,C 180,E1 -18243.001,E2 -18243.001} C_VEL
LIN {X 0,Y 263.188,Z 373.7,A -85,B 0,C 180,E1 -18246.386,E2 -18246.386} C_VEL
LIN {X 0,Y 263.267,Z 373.689,A -85,B 0,C 180,E1 -18249.692,E2 -18249.692} C_VEL
LIN {X 0,Y 263.354,Z 373.679,A -85,B 0,C 180,E1 -18254.52,E2 -18254.52} C_VEL
LIN {X 0,Y 263.358,Z 373.677,A -85,B 0,C 180,E1 -18259.232,E2 -18259.232} C_VEL
LIN {X 0,Y 263.56,Z 373.654,A -85,B 0,C 180,E1 -18262.336,E2 -18262.336} C_VEL
LIN {X 0,Y 263.754,Z 373.629,A -85,B 0,C 180,E1 -18268.471,E2 -18268.471} C_VEL
LIN {X 0,Y 263.753,Z 373.63,A -85,B 0,C 180,E1 -18271.525,E2 -18271.525} C_VEL
LIN {X 0,Y 263.573,Z 373.653,A -85,B 0,C 180,E1 -18277.66,E2 -18277.66} C_VEL
LIN {X 0,Y 263.373,Z 373.675,A -85,B 0,C 180,E1 -18280.764,E2 -18280.764} C_VEL
LIN {X 0,Y 263.35,Z 373.679,A -85,B 0,C 180,E1 -18285.476,E2 -18285.476} C_VEL
LIN {X 0,Y 263.261,Z 373.69,A -85,B 0,C 180,E1 -18290.305,E2 -18290.305} C_VEL
LIN {X 0,Y 263.206,Z 373.697,A -85,B 0,C 180,E1 -18295.289,E2 -18295.289} C_VEL
LIN {X 0,Y 263.172,Z 373.7,A -85,B 0,C 180,E1 -18298.728,E2 -18298.728} C_VEL
LIN {X 0,Y 263.13,Z 373.707,A -85,B 0,C 180,E1 -18302.286,E2 -18302.286} C_VEL
LIN {X 0,Y 263.186,Z 373.702,A -85,B 0,C 180,E1 -18305.976,E2 -18305.976} C_VEL
LIN {X 0,Y 263.156,Z 373.705,A -85,B 0,C 180,E1 -18309.861,E2 -18309.861} C_VEL
LIN {X 0,Y 263.185,Z 373.702,A -85,B 0,C 180,E1 -18313.968,E2 -18313.968} C_VEL
LIN {X 0,Y 263.208,Z 373.695,A -85,B 0,C 180,E1 -18318.383,E2 -18318.383} C_VEL
LIN {X 0,Y 263.199,Z 373.699,A -85,B 0,C 180,E1 -18323.229,E2 -18323.229} C_VEL
LIN {X 0,Y 263.176,Z 373.701,A -85,B 0,C 180,E1 -18325.889,E2 -18325.889} C_VEL
LIN {X 0,Y 263.145,Z 373.707,A -85,B 0,C 180,E1 -18329.506,E2 -18329.506} C_VEL
LIN {X 0,Y 263.188,Z 373.699,A -85,B 0,C 180,E1 -18333.002,E2 -18333.002} C_VEL
LIN {X 0,Y 263.175,Z 373.699,A -85,B 0,C 180,E1 -18336.386,E2 -18336.386} C_VEL
LIN {X 0,Y 263.255,Z 373.694,A -85,B 0,C 180,E1 -18339.693,E2 -18339.693} C_VEL
LIN {X 0,Y 263.342,Z 373.677,A -85,B 0,C 180,E1 -18344.522,E2 -18344.522} C_VEL
LIN {X 0,Y 263.365,Z 373.679,A -85,B 0,C 180,E1 -18349.234,E2 -18349.234} C_VEL
LIN {X 0,Y 263.564,Z 373.651,A -85,B 0,C 180,E1 -18352.338,E2 -18352.338} C_VEL
LIN {X 0,Y 263.746,Z 373.629,A -85,B 0,C 180,E1 -18358.473,E2 -18358.473} C_VEL
LIN {X 0,Y 263.744,Z 373.632,A -85,B 0,C 180,E1 -18361.527,E2 -18361.527} C_VEL
LIN {X 0,Y 263.565,Z 373.654,A -85,B 0,C 180,E1 -18367.662,E2 -18367.662} C_VEL
LIN {X 0,Y 263.366,Z 373.675,A -85,B 0,C 180,E1 -18370.766,E2 -18370.766} C_VEL
LIN {X 0,Y 263.342,Z 373.684,A -85,B 0,C 180,E1 -18375.479,E2 -18375.479} C_VEL
LIN {X 0,Y 263.255,Z 373.689,A -85,B 0,C 180,E1 -18380.308,E2 -18380.308} C_VEL
LIN {X 0,Y 263.184,Z 373.699,A -85,B 0,C 180,E1 -18384.248,E2 -18384.248} C_VEL
LIN {X 0,Y 262.54,Z 373.782,A -85,B 0,C 180,E1 -18385.527,E2 -18385.527} C_VEL
LIN {X 0,Y 259.638,Z 374.141,A -85,B 0,C 180,E1 -18387.608,E2 -18387.608} C_VEL
LIN {X 0,Y 257.169,Z 374.45,A -85,B 0,C 180,E1 -18389.301,E2 -18389.301} C_VEL
LIN {X 0,Y 256.135,Z 374.577,A -85,B 0,C 180,E1 -18390.616,E2 -18390.616} C_VEL
LIN {X 0,Y 256.066,Z 374.587,A -85,B 0,C 180,E1 -18391.062,E2 -18391.062} C_VEL
LIN {X 0,Y 256.115,Z 374.583,A -85,B 0,C 180,E1 -18395.188,E2 -18395.188} C_VEL
LIN {X 0,Y 256.14,Z 374.578,A -85,B 0,C 180,E1 -18399.13,E2 -18399.13} C_VEL
LIN {X 0,Y 256.136,Z 374.581,A -85,B 0,C 180,E1 -18403.312,E2 -18403.312} C_VEL
LIN {X 0,Y 256.157,Z 374.575,A -85,B 0,C 180,E1 -18407.798,E2 -18407.798} C_VEL
LIN {X 0,Y 256.105,Z 374.583,A -85,B 0,C 180,E1 -18410.867,E2 -18410.867} C_VEL
LIN {X 0,Y 256.171,Z 374.573,A -85,B 0,C 180,E1 -18414.824,E2 -18414.824} C_VEL
LIN {X 0,Y 256.225,Z 374.705,A -85,B 0,C 180,E1 -18415.677,E2 -18415.677} C_VEL
LIN {X 0,Y 259.522,Z 391.103,A -85,B 0,C 180,E1 -18420.829,E2 -18420.829} C_VEL
LIN {X 0,Y 260.149,Z 395.745,A -85,B 0,C 180,E1 -18422.226,E2 -18422.226} C_VEL
LIN {X 0,Y 258.938,Z 404.024,A -85,B 0,C 180,E1 -18424.587,E2 -18424.587} C_VEL
LIN {X 0,Y 259.925,Z 424.437,A -85,B 0,C 180,E1 -18425.544,E2 -18425.544} C_VEL
LIN {X 0,Y 262.651,Z 455.983,A -85,B 0,C 180,E1 -18427.05,E2 -18427.05} C_VEL
LIN {X 0,Y 260.461,Z 514.685,A -85,B 0,C 180,E1 -18429.673,E2 -18429.673} C_VEL
LIN {X 0,Y 259.662,Z 527.532,A -85,B 0,C 180,E1 -18430.536,E2 -18430.536} C_VEL
LIN {X 0,Y 258.729,Z 539.832,A -85,B 0,C 180,E1 -18431.656,E2 -18431.656} C_VEL
LIN {X 0,Y 257.742,Z 552.553,A -85,B 0,C 180,E1 -18433.161,E2 -18433.161} C_VEL
LIN {X 0,Y 256.891,Z 563.121,A -85,B 0,C 180,E1 -18434.735,E2 -18434.735} C_VEL
LIN {X 0,Y 256.146,Z 572.885,A -85,B 0,C 180,E1 -18436.515,E2 -18436.515} C_VEL
LIN {X 0,Y 255.565,Z 581.853,A -85,B 0,C 180,E1 -18438.502,E2 -18438.502} C_VEL
LIN {X 0,Y 255.21,Z 589.258,A -85,B 0,C 180,E1 -18440.491,E2 -18440.491} C_VEL
LIN {X 0,Y 255.084,Z 595.945,A -85,B 0,C 180,E1 -18442.688,E2 -18442.688} C_VEL
LIN {X 0,Y 255.083,Z 602.058,A -85,B 0,C 180,E1 -18445.261,E2 -18445.261} C_VEL
LIN {X 0,Y 255.141,Z 606.322,A -85,B 0,C 180,E1 -18447.634,E2 -18447.634} C_VEL
LIN {X 0,Y 255.154,Z 609.353,A -85,B 0,C 180,E1 -18450.002,E2 -18450.002} C_VEL
LIN {X 0,Y 254.838,Z 610.711,A -85,B 0,C 180,E1 -18451.582,E2 -18451.582} C_VEL
LIN {X 0,Y 254.578,Z 611.63,A -85,B 0,C 180,E1 -18453.167,E2 -18453.167} C_VEL
LIN {X 0,Y 254.332,Z 612.173,A -85,B 0,C 180,E1 -18455.846,E2 -18455.846} C_VEL
LIN {X 0,Y 254.319,Z 611.753,A -85,B 0,C 180,E1 -18457.944,E2 -18457.944} C_VEL
LIN {X 0,Y 254.544,Z 610.997,A -85,B 0,C 180,E1 -18459.537,E2 -18459.537} C_VEL
LIN {X 0,Y 254.954,Z 609.837,A -85,B 0,C 180,E1 -18461.127,E2 -18461.127} C_VEL
LIN {X 0,Y 255.54,Z 608.255,A -85,B 0,C 180,E1 -18462.712,E2 -18462.712} C_VEL
LIN {X 0,Y 257.627,Z 603.884,A -85,B 0,C 180,E1 -18465.833,E2 -18465.833} C_VEL
LIN {X 0,Y 259.549,Z 599.465,A -85,B 0,C 180,E1 -18468.145,E2 -18468.145} C_VEL
LIN {X 0,Y 262.223,Z 593.967,A -85,B 0,C 180,E1 -18470.392,E2 -18470.392} C_VEL
LIN {X 0,Y 265.374,Z 587.288,A -85,B 0,C 180,E1 -18472.584,E2 -18472.584} C_VEL
LIN {X 0,Y 269.066,Z 579.263,A -85,B 0,C 180,E1 -18474.705,E2 -18474.705} C_VEL
LIN {X 0,Y 273.305,Z 569.542,A -85,B 0,C 180,E1 -18476.746,E2 -18476.746} C_VEL
LIN {X 0,Y 278.104,Z 557.77,A -85,B 0,C 180,E1 -18478.697,E2 -18478.697} C_VEL
LIN {X 0,Y 282.099,Z 547.036,A -85,B 0,C 180,E1 -18480.093,E2 -18480.093} C_VEL
LIN {X 0,Y 286.587,Z 533.931,A -85,B 0,C 180,E1 -18481.409,E2 -18481.409} C_VEL
LIN {X 0,Y 290.219,Z 521.302,A -85,B 0,C 180,E1 -18482.399,E2 -18482.399} C_VEL
LIN {X 0,Y 293.612,Z 506.647,A -85,B 0,C 180,E1 -18483.303,E2 -18483.303} C_VEL
LIN {X 0,Y 300.418,Z 465.567,A -85,B 0,C 180,E1 -18485.182,E2 -18485.182} C_VEL
LIN {X 0,Y 300.918,Z 455.549,A -85,B 0,C 180,E1 -18486.133,E2 -18486.133} C_VEL
LIN {X 0,Y 301.028,Z 448.237,A -85,B 0,C 180,E1 -18487.007,E2 -18487.007} C_VEL
LIN {X 0,Y 299.805,Z 443.655,A -85,B 0,C 180,E1 -18488.314,E2 -18488.314} C_VEL
LIN {X 0,Y 298.88,Z 440.215,A -85,B 0,C 180,E1 -18489.484,E2 -18489.484} C_VEL
LIN {X 0,Y 297.487,Z 435.069,A -85,B 0,C 180,E1 -18491.838,E2 -18491.838} C_VEL
LIN {X 0,Y 296.661,Z 432.178,A -85,B 0,C 180,E1 -18494.461,E2 -18494.461} C_VEL
LIN {X 0,Y 296.825,Z 430.861,A -85,B 0,C 180,E1 -18496.635,E2 -18496.635} C_VEL
LIN {X 0,Y 297.717,Z 430.719,A -85,B 0,C 180,E1 -18498.787,E2 -18498.787} C_VEL
LIN {X 0,Y 299.716,Z 432.897,A -85,B 0,C 180,E1 -18501.52,E2 -18501.52} C_VEL
LIN {X 0,Y 301.67,Z 436.029,A -85,B 0,C 180,E1 -18503.394,E2 -18503.394} C_VEL
LIN {X 0,Y 303.861,Z 439.753,A -85,B 0,C 180,E1 -18505.05,E2 -18505.05} C_VEL
LIN {X 0,Y 296.409,Z 483.855,A -85,B 0,C 180,E1 -18507.104,E2 -18507.104} C_VEL
LIN {X 0,Y 293.64,Z 497.816,A -85,B 0,C 180,E1 -18508.025,E2 -18508.025} C_VEL
LIN {X 0,Y 290.672,Z 509.837,A -85,B 0,C 180,E1 -18509.083,E2 -18509.083} C_VEL
LIN {X 0,Y 286.974,Z 522.192,A -85,B 0,C 180,E1 -18510.471,E2 -18510.471} C_VEL
LIN {X 0,Y 283.482,Z 532.303,A -85,B 0,C 180,E1 -18511.898,E2 -18511.898} C_VEL
LIN {X 0,Y 279.057,Z 543.35,A -85,B 0,C 180,E1 -18513.849,E2 -18513.849} C_VEL
LIN {X 0,Y 274.94,Z 552.293,A -85,B 0,C 180,E1 -18515.858,E2 -18515.858} C_VEL
LIN {X 0,Y 271.255,Z 559.566,A -85,B 0,C 180,E1 -18517.933,E2 -18517.933} C_VEL
LIN {X 0,Y 267.987,Z 565.448,A -85,B 0,C 180,E1 -18520.066,E2 -18520.066} C_VEL
LIN {X 0,Y 265.027,Z 570.147,A -85,B 0,C 180,E1 -18522.244,E2 -18522.244} C_VEL
LIN {X 0,Y 261.975,Z 574.405,A -85,B 0,C 180,E1 -18524.971,E2 -18524.971} C_VEL
LIN {X 0,Y 259.645,Z 576.997,A -85,B 0,C 180,E1 -18527.494,E2 -18527.494} C_VEL
LIN {X 0,Y 257.446,Z 578.598,A -85,B 0,C 180,E1 -18530.573,E2 -18530.573} C_VEL
LIN {X 0,Y 256.652,Z 578.753,A -85,B 0,C 180,E1 -18532.13,E2 -18532.13} C_VEL
LIN {X 0,Y 256.122,Z 578.487,A -85,B 0,C 180,E1 -18533.698,E2 -18533.698} C_VEL
LIN {X 0,Y 255.644,Z 577.834,A -85,B 0,C 180,E1 -18535.269,E2 -18535.269} C_VEL
LIN {X 0,Y 255.13,Z 576.791,A -85,B 0,C 180,E1 -18536.842,E2 -18536.842} C_VEL
LIN {X 0,Y 254.72,Z 575.285,A -85,B 0,C 180,E1 -18538.419,E2 -18538.419} C_VEL
LIN {X 0,Y 254.466,Z 572.218,A -85,B 0,C 180,E1 -18540.791,E2 -18540.791} C_VEL
LIN {X 0,Y 254.553,Z 568.091,A -85,B 0,C 180,E1 -18543.165,E2 -18543.165} C_VEL
LIN {X 0,Y 254.691,Z 562.769,A -85,B 0,C 180,E1 -18545.542,E2 -18545.542} C_VEL
LIN {X 0,Y 255.143,Z 554.897,A -85,B 0,C 180,E1 -18548.315,E2 -18548.315} C_VEL
LIN {X 0,Y 255.685,Z 546.304,A -85,B 0,C 180,E1 -18550.692,E2 -18550.692} C_VEL
LIN {X 0,Y 256.363,Z 537.622,A -85,B 0,C 180,E1 -18552.669,E2 -18552.669} C_VEL
LIN {X 0,Y 257.273,Z 527.134,A -85,B 0,C 180,E1 -18554.636,E2 -18554.636} C_VEL
LIN {X 0,Y 258.172,Z 515.439,A -85,B 0,C 180,E1 -18556.405,E2 -18556.405} C_VEL
LIN {X 0,Y 259.035,Z 503.077,A -85,B 0,C 180,E1 -18557.901,E2 -18557.901} C_VEL
LIN {X 0,Y 259.928,Z 488.654,A -85,B 0,C 180,E1 -18559.24,E2 -18559.24} C_VEL
LIN {X 0,Y 260.615,Z 473.97,A -85,B 0,C 180,E1 -18560.213,E2 -18560.213} C_VEL
LIN {X 0,Y 263.499,Z 399.16,A -85,B 0,C 180,E1 -18563.468,E2 -18563.468} C_VEL
LIN {X 0,Y 256.236,Z 374.836,A -85,B 0,C 180,E1 -18564.866,E2 -18564.866} C_VEL
LIN {X 0,Y 256.195,Z 374.569,A -85,B 0,C 180,E1 -18564.966,E2 -18564.966} C_VEL
LIN {X 0,Y 256.12,Z 374.579,A -85,B 0,C 180,E1 -18569.599,E2 -18569.599} C_VEL
LIN {X 0,Y 256.082,Z 374.582,A -85,B 0,C 180,E1 -18573.291,E2 -18573.291} C_VEL
LIN {X 0,Y 256.121,Z 374.579,A -85,B 0,C 180,E1 -18577.27,E2 -18577.27} C_VEL
LIN {X 0,Y 256.059,Z 374.585,A -85,B 0,C 180,E1 -18581.202,E2 -18581.202} C_VEL
LIN {X 0,Y 256.062,Z 374.587,A -85,B 0,C 180,E1 -18585.529,E2 -18585.529} C_VEL
LIN {X 0,Y 256.059,Z 374.586,A -85,B 0,C 180,E1 -18588.795,E2 -18588.795} C_VEL
LIN {X 0,Y 256.143,Z 374.576,A -85,B 0,C 180,E1 -18592.868,E2 -18592.868} C_VEL
LIN {X 0,Y 256.08,Z 374.584,A -85,B 0,C 180,E1 -18596.707,E2 -18596.707} C_VEL
LIN {X 0,Y 256.138,Z 374.576,A -85,B 0,C 180,E1 -18601.405,E2 -18601.405} C_VEL
LIN {X 0,Y 256.171,Z 374.574,A -85,B 0,C 180,E1 -18605.698,E2 -18605.698} C_VEL
LIN {X 0,Y 256.17,Z 374.571,A -85,B 0,C 180,E1 -18609.103,E2 -18609.103} C_VEL
LIN {X 0,Y 256.303,Z 374.56,A -85,B 0,C 180,E1 -18614.084,E2 -18614.084} C_VEL
LIN {X 0,Y 256.3,Z 374.556,A -85,B 0,C 180,E1 -18618.932,E2 -18618.932} C_VEL
LIN {X 0,Y 256.518,Z 374.533,A -85,B 0,C 180,E1 -18622.125,E2 -18622.125} C_VEL
LIN {X 0,Y 256.502,Z 374.53,A -85,B 0,C 180,E1 -18626.857,E2 -18626.857} C_VEL
LIN {X 0,Y 256.775,Z 374.502,A -85,B 0,C 180,E1 -18629.998,E2 -18629.998} C_VEL
LIN {X 0,Y 256.502,Z 374.53,A -85,B 0,C 180,E1 -18633.139,E2 -18633.139} C_VEL
LIN {X 0,Y 256.541,Z 374.53,A -85,B 0,C 180,E1 -18637.871,E2 -18637.871} C_VEL
LIN {X 0,Y 256.309,Z 374.555,A -85,B 0,C 180,E1 -18641.064,E2 -18641.064} C_VEL
LIN {X 0,Y 256.299,Z 374.561,A -85,B 0,C 180,E1 -18645.913,E2 -18645.913} C_VEL
LIN {X 0,Y 256.165,Z 374.572,A -85,B 0,C 180,E1 -18650.893,E2 -18650.893} C_VEL
LIN {X 0,Y 256.186,Z 374.571,A -85,B 0,C 180,E1 -18655.137,E2 -18655.137} C_VEL
LIN {X 0,Y 256.107,Z 374.583,A -85,B 0,C 180,E1 -18659.598,E2 -18659.598} C_VEL
LIN {X 0,Y 256.081,Z 374.584,A -85,B 0,C 180,E1 -18663.288,E2 -18663.288} C_VEL
LIN {X 0,Y 256.136,Z 374.578,A -85,B 0,C 180,E1 -18667.277,E2 -18667.277} C_VEL
LIN {X 0,Y 256.117,Z 374.579,A -85,B 0,C 180,E1 -18671.188,E2 -18671.188} C_VEL
LIN {X 0,Y 256.111,Z 374.581,A -85,B 0,C 180,E1 -18674.482,E2 -18674.482} C_VEL
LIN {X 0,Y 256.127,Z 374.576,A -85,B 0,C 180,E1 -18678.811,E2 -18678.811} C_VEL
LIN {X 0,Y 256.148,Z 374.576,A -85,B 0,C 180,E1 -18682.871,E2 -18682.871} C_VEL
LIN {X 0,Y 256.077,Z 374.582,A -85,B 0,C 180,E1 -18686.709,E2 -18686.709} C_VEL
LIN {X 0,Y 256.134,Z 374.58,A -85,B 0,C 180,E1 -18691.402,E2 -18691.402} C_VEL
LIN {X 0,Y 256.159,Z 374.576,A -85,B 0,C 180,E1 -18695.698,E2 -18695.698} C_VEL
LIN {X 0,Y 256.158,Z 374.575,A -85,B 0,C 180,E1 -18699.104,E2 -18699.104} C_VEL
LIN {X 0,Y 256.291,Z 374.556,A -85,B 0,C 180,E1 -18704.085,E2 -18704.085} C_VEL
LIN {X 0,Y 256.301,Z 374.557,A -85,B 0,C 180,E1 -18708.934,E2 -18708.934} C_VEL
LIN {X 0,Y 256.531,Z 374.527,A -85,B 0,C 180,E1 -18712.127,E2 -18712.127} C_VEL
LIN {X 0,Y 256.709,Z 374.506,A -85,B 0,C 180,E1 -18718.431,E2 -18718.431} C_VEL
LIN {X 0,Y 256.707,Z 374.508,A -85,B 0,C 180,E1 -18721.569,E2 -18721.569} C_VEL
LIN {X 0,Y 256.532,Z 374.529,A -85,B 0,C 180,E1 -18727.873,E2 -18727.873} C_VEL
LIN {X 0,Y 256.302,Z 374.556,A -85,B 0,C 180,E1 -18731.067,E2 -18731.067} C_VEL
LIN {X 0,Y 256.291,Z 374.559,A -85,B 0,C 180,E1 -18735.916,E2 -18735.916} C_VEL
LIN {X 0,Y 256.159,Z 374.574,A -85,B 0,C 180,E1 -18740.896,E2 -18740.896} C_VEL
LIN {X 0,Y 256.18,Z 374.575,A -85,B 0,C 180,E1 -18745.139,E2 -18745.139} C_VEL
LIN {X 0,Y 256.096,Z 374.584,A -85,B 0,C 180,E1 -18749.602,E2 -18749.602} C_VEL
LIN {X 0,Y 256.066,Z 374.587,A -85,B 0,C 180,E1 -18751.062,E2 -18751.062} C_VEL
LIN {X 0,Y 255.442,Z 374.671,A -85,B 0,C 180,E1 -18752.375,E2 -18752.375} C_VEL
